		// State Change Condition
		IF (SIf.stErr.bolComError = TRUE) OR ((SIf.stErr.bolRFIDError = TRUE) AND (udiJobCount > SIf.stCfg.udiRetry)) THEN
			stStateMachine.intStateNext := cRFD_STA_Error;
		ELSIF (SIf.stErr.bolRFIDError = TRUE) THEN
			udiJobCount := udiJobCount + 1;
			stStateMachine.intStateLastCycle := 0; // Startcycle again
		ELSIF (stSubStateMachine.intState = cRFD_SUB_SubStatesEnd) THEN
			udiJobCount := 0;
			stStateMachine.intStateNext := cRFD_STA_WaitForJob;
		END_IF
		
	END_IF

//--------------------------------------------------------------------------------------
// Exit action
	IF (stStateMachine.intState<>stStateMachine.intStateNext) THEN
		SIf.intCmd := cRFD_CMD_DONE;
	END_IF
END_METHOD

METHOD PROTECTED sta_TagInitBusy : BOOL
// state implemetation
//--------------------------------------------------------------------------------------
// Entry action
	IF (stStateMachine.intState<>stStateMachine.intStateLastCycle) THEN
		stStateMachine.intStateLastCycle := stStateMachine.intState;
		
	END_IF


//--------------------------------------------------------------------------------------
// Cyclic action
	IF (stStateMachine.intState=stStateMachine.intStateLastCycle) THEN

		
		// State Change Condition
		IF (FALSE) THEN
			stStateMachine.intStateNext := cRFD_STA_Error;
		ELSIF (TRUE) THEN
			stStateMachine.intStateNext := cRFD_STA_WaitForJob;
		END_IF
		
	END_IF

//--------------------------------------------------------------------------------------
// Exit action
	IF (stStateMachine.intState<>stStateMachine.intStateNext) THEN
		IF SIf.intCmd = stStateMachine.intState THEN
			SIf.intCmd := cRFD_CMD_DONE;
		END_IF
	END_IF
END_METHOD

METHOD PROTECTED sta_WaitForJob : BOOL
// state implemetation
//--------------------------------------------------------------------------------------
// Entry action
	IF (stStateMachine.intState<>stStateMachine.intStateLastCycle) THEN
		stStateMachine.intStateLastCycle := stStateMachine.intState;
		
	END_IF


//--------------------------------------------------------------------------------------
// Cyclic action
	IF (stStateMachine.intState=stStateMachine.intStateLastCycle) THEN

		
		// State Change Condition
		IF (FALSE) THEN
			stStateMachine.intStateNext := cRFD_STA_Error;
		ELSIF (SIf.intCmd=cRFD_CMD_Read) THEN
			stStateMachine.intStateNext := cRFD_STA_ReadBusy;
		ELSIF (SIf.intCmd=cRFD_CMD_CTRL_ON) THEN
			stStateMachine.intStateNext := cRFD_STA_PowerOnBusy;
		ELSIF (SIf.intCmd=cRFD_CMD_Write) THEN
			stStateMachine.intStateNext := cRFD_STA_WriteBusy;
		ELSIF (SIf.intCmd=cRFD_CMD_MDS) THEN
			stStateMachine.intStateNext := cRFD_STA_MDSBusy;
		ELSIF (SIf.intCmd=cRFD_CMD_SLG) THEN
			stStateMachine.intStateNext := cRFD_STA_SLGBusy;
		ELSIF (SIf.intCmd=cRFD_CMD_CTRL_OFF) THEN
			stStateMachine.intStateNext := cRFD_STA_OFFBusy;
		ELSIF (SIf.intCmd=cRFD_STA_CheckBusy) THEN
			stStateMachine.intStateNext := cRFD_STA_CheckBusy;
		END_IF
		
	END_IF

//--------------------------------------------------------------------------------------
// Exit action
	IF (stStateMachine.intState<>stStateMachine.intStateNext) THEN
		;
	END_IF
END_METHOD

METHOD PROTECTED sta_WriteBusy : BOOL
// state implemetation
//--------------------------------------------------------------------------------------
// Entry action
	IF (stStateMachine.intState<>stStateMachine.intStateLastCycle) THEN
			stStateMachine.intStateLastCycle := stStateMachine.intState;
			// Byte 0 => Lenght
			aTxData[0] := 5 + SIf.stCur.usiCount;
			// Byte 1 => Command write 1=single; 11=continious
			aTxData[1] := 1;
			// Byte 2 => Spare
			aTxData[2] := 0;
			// Byte 3 => Adress MSB
			uinValue := SIf.stCur.uinAdressTag;
			uinValue := ROL(uinValue,8);
			aTxData[3] := UINT_TO_USINT(uinValue);
			// Byte 4 => Adress LSB
			aTxData[4] := UINT_TO_USINT(SIf.stCur.uinAdressTag);
			// Byte 5 =>Lenght
			aTxData[5] := SIf.stCur.usiCount;
 
			IF ((SIf.stCur.uinAdressData+SIf.stCur.usiCount <= 255) AND (SIf.stCur.usiCount+6 <= 255)) THEN
				FOR udiLoopBuffer := 0 TO (SIf.stCur.usiCount) DO
					aTxData[udiLoopBuffer+6] := SIf.stCur.pData^[SIf.stCur.uinAdressData+udiLoopBuffer];
				END_FOR	
				udiComSizeSendData := SIf.stCur.usiCount+6;
				bolComSend := TRUE;		
			ELSE
				SIf.stErr.bolComError := TRUE;
			END_IF
							
	END_IF


//--------------------------------------------------------------------------------------
// Cyclic action
	IF (stStateMachine.intState=stStateMachine.intStateLastCycle) THEN
		
		// State Change Condition
		IF (SIf.stErr.bolComError = TRUE) OR ((SIf.stErr.bolRFIDError = TRUE) AND (udiJobCount > SIf.stCfg.udiRetry)) THEN
			stStateMachine.intStateNext := cRFD_STA_Error;
		ELSIF (SIf.stErr.bolRFIDError = TRUE) THEN
			udiJobCount := udiJobCount + 1;
			stStateMachine.intStateLastCycle := 0; // Startcycle again
		ELSIF ((SIf.stErr.bolComError = 0) AND (bolWriteDone = TRUE)) THEN
			bolWriteDone := FALSE;
			udiJobCount := 0;
			stStateMachine.intStateNext := cRFD_STA_WaitForJob;
		END_IF
	
	END_IF

//--------------------------------------------------------------------------------------
// Exit action
	IF (stStateMachine.intState<>stStateMachine.intStateNext) THEN
		SIf.intCmd := cRFD_CMD_DONE;
	END_IF
END_METHOD

METHOD PROTECTED StateMachine : BOOL

// main statemachine of base controller
CASE stStateMachine.intState OF
	cRFD_STA_OffBusy: 
        THIS^.sta_OffBusy();
	cRFD_STA_Off: 
        THIS^.sta_Off();
    cRFD_STA_PowerOnBusy: 
        THIS^.sta_PowerOnBusy();
	cRFD_STA_WaitForJob: 
        THIS^.sta_WaitForJob();
	cRFD_STA_WriteBusy: 
        THIS^.sta_WriteBusy();
    cRFD_STA_ReadBusy: 
        THIS^.sta_ReadBusy();
	cRFD_STA_TagInitBusy: 
        THIS^.sta_TagInitBusy();
	cRFD_STA_CheckBusy: 
        THIS^.sta_CheckBusy();
	cRFD_STA_MDSBusy: 
        THIS^.sta_MDSBusy();
	cRFD_STA_SLGBusy: 
        THIS^.sta_SLGBusy();
    cRFD_STA_Error: 
        THIS^.sta_Error();
END_CASE;
END_METHOD

METHOD PROTECTED StateMachine_Service : BOOL


// main statemachine of base controller
CASE SIf.intServiceCmd OF
//	cRFD_CMD_MDS: 
//		THIS^.sJobWriteParameter();
//	cYAD_SCMD_READ_PARA: 
//		THIS^.sJobReadParameter();
//	cYAD_SCMD_RESET_ABSENCODER: 
//		THIS^.sJobAbsEncReset();
ELSE
	usiCaseScmd := 0;
	

	
END_CASE;
END_METHOD

END_FUNCTION_BLOCK

// POUs/Controller/Driver/RFD (RFID Driver)/FB_RFR
FUNCTION_BLOCK FB_RFR
VAR
	bolActivate: BOOL := TRUE;
	bolInitDone: BOOL;
	bolInitComDone: BOOL;
	///Communication sending is busy to the serial Card
	bolComSend: BOOL;
	/// Size of Sendingdata
	udiComSizeSendData: UDINT;
	///Communication Data Received
	bolComDataReceived: BOOL;
	/// Size of received Data from serial interface
	udiComSizeReceiveData: UDINT;
	///Sdo Setting is busy to the serial Card
	bolSdoBusy: BOOL;
	///Sdo Setting executing
	bolSdoExecute: BOOL;
	/// Job Reading is done
	bolReadDone: BOOL;
	/// Job Writing is done
	bolWriteDone: BOOL;
	/// Job Reset SLG is done
	bolResetJobDone: BOOL;
	/// Job Reset SLG has Error
	bolResetJobError: BOOL;
	/// Information to SDO Error
	udiSdoErrorNbr: UDINT;
	/// Information to Error
	udiComErrorNbr: UDINT;
	/// Count Reset cycles
	udiResetCount: UDINT;
	/// Count Job Tryals
	udiJobCount: UDINT;
	/// State information from RF ID Tag
	bytRFIDState: BYTE;
	/// BCC Calculation
	bytCheckValue: BYTE;
	/// driver specific interface
	SIf: T_RFD;
	/// get direct Buffer from Interface
	/// access over mapping!! {attribute 'TcLinkTo':='TIID^Device 1 (EtherCAT)^Box 1 (SGDV-E1 CoE Drive)^2nd Transmit PDO mapping^Status word'}
	aRxData: ARRAY[0..255] OF BYTE;
	aTxData: ARRAY[0..255] OF BYTE;
	/// Function for serial communication
	fbEcCoeSdoWrite: TC2_ETHERCAT.FB_EcCoESdoWrite;
	fbExCom: FB_ExCom;
	stStateMachine: T_RFD_StateMachine;
	stSubStateMachine: T_RFD_StateMachine;
	///case variable
	usiCase: USINT;
	///case variable for service cmd's
	usiCaseScmd: USINT;
	/// help values for parameter handling
	sinValue: SINT;
	intValue: INT;
	dinValue: DINT;
	usiValue: USINT;
	uinValue: UINT;
	udiValue: UDINT;
	uliValue: ULINT;
	pTemp: POINTER TO ARRAY[0..7] OF BYTE;
	strTemp: STRING(18);
	udiI: UDINT;
	udiLoopBuffer: UDINT;
	udiLoopData: UDINT;
	udiLoopSend: UDINT;
END_VAR

(*__________________________________________________________________________________________________
¦	
¦	Vistaprint Schweiz GmbH
¦	CH - 8401 Winterthur
¦
¦	www.vistaprint.ch - info@vistaprint.ch
¦___________________________________________________________________________________________________

Function desription:
Driver for Simatic RFID Reader RF382R 6GT2801-3AB20-0AX0 (only read function)


History:
Version		Date			Author		Comment
---------------------------------------------------------------------------------------------------
0.00.1		09.07.2013		AVME/PRE	Start history
0.00.2		18.09.2013		AVME/KVO	no initial write of parameter to RFID reader at PowerOnBusy
0.00.3		25.09.2013		AVME/KVO	always set sample error and go to error state!
___________________________________________________________________________________________________*)


IF (bolActivate) THEN // cyclic call enabled
	
	IF (bolInitDone=FALSE) THEN // first cycle -> init
		CtrlInit();
		bolInitDone := TRUE;
	ELSE
		CycleStartDuty();
		
		StateMachine_Service(); // handles asynchron service commands
		
		StateMachine();
		
		CycleEndDuty();
	END_IF
	
END_IF;

METHOD PROTECTED CtrlInit : BOOL
// one time first cyclic call
;
END_METHOD

METHOD PROTECTED CycleEndDuty : BOOL
SIf.strState := THIS^.getCmdState(intCmdState:=stStateMachine.intState,bolState:=TRUE);

IF (stStateMachine.intState<>stStateMachine.intStateNext) THEN
	stStateMachine.intState := stStateMachine.intStateNext;  // set next state for next cycle
END_IF

(***************************************************************
        Function Block Calls
***************************************************************)
END_METHOD

METHOD PROTECTED CycleStartDuty : BOOL
// ----------------------------------------------------------------------------------
// cyclic actions outside of statemachine
fbExCom(
	In_pRxData:= ADR(aRxData), 
	In_pTxData:= ADR(aTxData), 
	In_udiTxCount:= udiComSizeSendData, 
	In_bolErrorAck:= SIf.stErr.bolErrAck, 
	InOut_bolSend:= bolComSend, 
	InOut_bolRec:= bolComDataReceived, 
	Out_udiRxCount=> udiComSizeReceiveData, 
	Out_bolComError=> SIf.stErr.bolComError, 
	Out_bolProtocolErr=> SIf.stErr.bolProtcolError, 
	Out_udiErrorCode=> udiComErrorNbr);

(* program code at the beginning of each PLC cycle *)
IF bolInitComDone=TRUE THEN
	// Received Data checking and interpreting
	IF bolComDataReceived = TRUE THEN
		IF (aRxData[0] = 1) AND (udiComSizeReceiveData = 3) THEN		// Ack Reset
			IF aRxData[1] = 0 THEN
				bolResetJobDone := TRUE;
			ELSE
				 SIf.stErr.bolProtcolError := TRUE;
			END_IF
		ELSE
			// UID
			MEMCPY(destAddr:=ADR(strTemp), srcAddr:=ADR(aRxData[0]), n:=16);

			uliValue := FB_HEXSTRING_TO_ULINT(in_strSTRING:= strTemp);
			pTemp := ADR(SIf.stStatus.abyteUID[0]);
			MEMCPY(destAddr:=ADR(SIf.stStatus.abyteUID[0]), srcAddr:=ADR(uliValue), n:=8);		// COPY to ID 
			
		END_IF
		bolComDataReceived := FALSE;
	END_IF
END_IF

// always go to Error 
IF ((SIf.stErr.bolProtcolError) OR  (SIf.stErr.bolRFIDError) OR (SIf.stErr.bolSDOError)) THEN
	SIf.stErr.bolErrorActive := TRUE; // set sample Error -> got to Error state
END_IF

IF (SIf.stErr.bolErrorActive) AND (stStateMachine.intState<>cRFD_STA_Error)  THEN
	stStateMachine.intStateNext := cRFD_STA_Error;
ELSIF (stStateMachine.intState<cRFD_STA_PowerOnBusy) AND (stStateMachine.intState<>cRFD_STA_Error) THEN
	stStateMachine.intStateNext := cRFD_STA_PowerOnBusy;
END_IF

SIf.strCmd := THIS^.getCmdState(intCmdState:=SIf.intCmd,bolState:=FALSE);
END_METHOD

METHOD FB_init : BOOL
VAR_INPUT
	///if TRUE, the retain variables are initialized (warm start / cold start)
	bInitRetains: BOOL;
	///if TRUE, the instance afterwards gets moved into the copy code (online change)
	bInCopyCode: BOOL;
END_VAR
VAR
	udiTaskCnt: UDINT;
	ii: UINT;
END_VAR
SIf.intCmd := cRFD_CMD_DONE;
SIf.intServiceCmd := cRFD_CMD_DONE; // not used at the moment
stStateMachine.intStateLastCycle  := cRFD_CMD_DONE; //EntryStop of power BASE_PLC.OFF enable

// Communication Settings
SIf.stCfg.eTyp := E_Typ_RFW.RF382R;
SIf.stCfg.uinBaudrate := INT_TO_USINT(E_Typ_Baudrate.baud_38400);
SIf.stCfg.stNetId := '192.168.70.26.3.1';
SIf.stCfg.uinSlaveAddr := 1002;
END_METHOD

METHOD PROTECTED getCmdState : STRING
VAR_INPUT
	intCmdState: INT;
	bolState: BOOL;
END_VAR
// get string cmd/state string information in runtime
IF (bolState=FALSE) THEN
	// cmd's
	CASE intCmdState OF
		cRFD_CMD_DONE: 
			getCmdState := 'cRFD_CMD_DONE';
		cRFD_CMD_CTRL_ON: 
			getCmdState := 'cRFD_CMD_CTRL_ON';

	END_CASE;
ELSE

// States
	CASE intCmdState OF
		cRFD_STA_Error: 
			getCmdState := 'cRFD_STA_Error';
		cRFD_STA_WaitForJob: 
			getCmdState := 'cRFD_STA_WaitForJob';
		cRFD_STA_PowerOnBusy: 
			getCmdState := 'cRFD_STA_PowerOnBusy';

	END_CASE;
END_IF
END_METHOD

METHOD getSIf : POINTER TO T_RFD
getSIf := ADR(SIf);
END_METHOD

METHOD PROTECTED sta_Error : BOOL
// state implemetation
//--------------------------------------------------------------------------------------
// Entry action
	IF (stStateMachine.intState<>stStateMachine.intStateLastCycle) THEN
		stStateMachine.intStateHistory := stStateMachine.intStateLastCycle;
		stStateMachine.intStateLastCycle := stStateMachine.intState;
		
	END_IF


//--------------------------------------------------------------------------------------
// Cyclic action
	IF (stStateMachine.intState=stStateMachine.intStateLastCycle) THEN
		SIf.stErr.bolErrorActive := TRUE;
		IF (SIf.stErr.bolComError = TRUE) OR (SIf.stErr.bolProtcolError = TRUE) THEN
			SIf.stErr.udiErrorID := udiComErrorNbr;
		ELSIF SIf.stErr.bolSDOError = TRUE THEN
			SIf.stErr.udiErrorID := udiSdoErrorNbr;
		ELSIF (udiResetCount >=SIf.stCfg.udiRetry) OR (udiJobCount >= SIf.stCfg.udiRetry) THEN
			SIf.stErr.udiErrorID := SIf.stCfg.udiRetry;
		ELSE
			SIf.stErr.udiErrorID := 0;
		END_IF

		
		// State Change Condition
		IF (SIf.stErr.bolErrAck = TRUE) THEN
			// Reset all active errors
			SIf.stErr.bolErrorActive := FALSE;
			SIf.stErr.bolComError := FALSE;
			SIf.stErr.bolProtcolError := FALSE;
			SIf.stErr.bolSDOError := FALSE;
			SIf.stErr.udiErrorID := 0;
			stStateMachine.intStateNext := cRFD_STA_PowerOnBusy;		
		END_IF
	END_IF




//--------------------------------------------------------------------------------------
// Exit action
	IF (stStateMachine.intState<>stStateMachine.intStateNext) THEN
		;
	END_IF
END_METHOD

METHOD PROTECTED sta_PowerOnBusy : BOOL
// state implemetation
//--------------------------------------------------------------------------------------
// Entry action
	IF (stStateMachine.intState<>stStateMachine.intStateLastCycle) THEN
		stStateMachine.intStateLastCycle := stStateMachine.intState;
			//IF bolInitComDone=FALSE THEN
				// direct write parameter doesn't work!! KVO 17.09.2013 with new Kannegiesser RFID
				// Feedback rx[0..2] 255 4 251 -> Baudrate/task time not 2ms
				// no Feedback -> parameter set? estimated  rx[0..2] 1 0 1
				// decision with Rolf Engelputzeder 18.09.2013 
				// don't use write parameter at the moment:
				stSubStateMachine.intState := cRFD_SUB_SubStatesEnd;// cRFD_SUB_ClearBuffer;		// First Time set Baudrate and communication Settings
				stSubStateMachine.intStateNext := cRFD_SUB_SubStatesEnd;// cRFD_SUB_ClearBuffer;		// First Time set Baudrate and communication Settings
				bolInitComDone := TRUE; // old without this condition
				
				(*
				// original set parameter to RFID
				stSubStateMachine.intState := cRFD_SUB_ClearBuffer;		// First Time set Baudrate and communication Settings
				stSubStateMachine.intStateNext := cRFD_SUB_ClearBuffer;
				*)
			//END_IF
			bolSdoExecute := FALSE;
			bolResetJobDone := FALSE;
	END_IF


//--------------------------------------------------------------------------------------
// Cyclic action
	IF (stStateMachine.intState=stStateMachine.intStateLastCycle) THEN
		
		// main statemachine of base controller
		CASE stSubStateMachine.intState OF
			cRFD_SUB_SetBaudrate:
				IF stSubStateMachine.intStateLastCycle <> stSubStateMachine.intState THEN
					stSubStateMachine.intStateLastCycle := stSubStateMachine.intState;
				END_IF
				fbEcCoeSdoWrite(
					sNetId:= SIf.stCfg.stNetId, 
					nSlaveAddr:= SIf.stCfg.uinSlaveAddr, 
					nIndex:= SIf.stCfg.uinCoeIndexComSettings, 
					nSubIndex:= SIf.stCfg.usiCoeSubindexComBaudrate, 
					pSrcBuf:= ADR(SIf.stCfg.uinBaudrate), 
					cbBufLen:= SIZEOF(SIf.stCfg.uinBaudrate), 
					bExecute:= bolSdoExecute, 
					tTimeout:= DEFAULT_ADS_TIMEOUT, 
					bBusy=> bolSdoBusy, 
					bError=> SIf.stErr.bolSDOError, 
					nErrId=> udiSdoErrorNbr);
					
					
				IF 	(bolSdoExecute = TRUE) THEN
					IF ((SIf.stErr.bolSDOError = FALSE) AND (bolSdoBusy = FALSE)) THEN
						bolSdoExecute := FALSE;
						stSubStateMachine.intStateNext := cRFD_SUB_ClearBuffer;
					END_IF
				ELSE
					bolSdoExecute := TRUE;
				END_IF
				
			
			cRFD_SUB_SetComSettings:
				IF stSubStateMachine.intStateLastCycle <> stSubStateMachine.intState THEN
					stSubStateMachine.intStateLastCycle := stSubStateMachine.intState;
				END_IF
				fbEcCoeSdoWrite(
					sNetId:= SIf.stCfg.stNetId, 
					nSlaveAddr:= SIf.stCfg.uinSlaveAddr, 
					nSubIndex:= SIf.stCfg.usiCoeSubindexComDataframe, 
					nIndex:= SIf.stCfg.uinCoeIndexComSettings, 
					pSrcBuf:= ADR(SIf.stCfg.uinComSettings), 
					cbBufLen:= SIZEOF(SIf.stCfg.uinComSettings), 
					bExecute:= bolSdoExecute, 
					tTimeout:= T#2S, 
					bBusy=> bolSdoBusy, 
					bError=> SIf.stErr.bolSDOError, 
					nErrId=> udiSdoErrorNbr);
					
				IF 	(bolSdoExecute = TRUE) THEN
					IF ((SIf.stErr.bolSDOError = FALSE) AND (bolSdoBusy = FALSE)) THEN
						bolSdoExecute := FALSE;
						stSubStateMachine.intStateNext := cRFD_SUB_ClearBuffer;
					END_IF
				ELSE
					bolSdoExecute := TRUE;
				END_IF

	
			cRFD_SUB_ClearBuffer: 	 
				IF stSubStateMachine.intStateLastCycle <> stSubStateMachine.intState THEN
					stSubStateMachine.intStateLastCycle := stSubStateMachine.intState;
				END_IF
				bolInitComDone := TRUE;
				IF (SIf.stErr.bolComError = FALSE) THEN
					stSubStateMachine.intStateNext := cRFD_SUB_InitString;
				END_IF

				
			cRFD_SUB_InitString: 
				IF stSubStateMachine.intStateLastCycle <> stSubStateMachine.intState THEN
					stSubStateMachine.intStateLastCycle := stSubStateMachine.intState;
					// Byte 0 => Para = 16#01
					aTxData[0] := 1;
					// Byte 1 => Memory
					aTxData[1] := SIf.stCfg.usiMemory;
					// Byte 2 => Spare
					aTxData[2] := 0;
					// Byte 3 => Spare
					aTxData[3] := 0;
					// Byte 4 => Spare
					aTxData[4] := 0;
					// Byte 5 => Spare
					aTxData[5] := 0;
					// Byte 6 => Spare
					aTxData[6] := 0;
					// Byte 7 => Scan Mode
					aTxData[7] := SIf.stCfg.usiScanMode;
					// Byte 8 => Lock Time High Byte
					aTxData[8] := UINT_TO_BYTE(SIf.stCfg.uinLockTime_ms/100);
					// Byte 9 => Lock Time Low Byte
					aTxData[9] := UINT_TO_BYTE(SHR((SIf.stCfg.uinLockTime_ms/100),8));
					// Byte 10 => Spare
					aTxData[10] := 0;
					// Byte 11 => Spare
					aTxData[11] := 0;
					// Byte 12 => Spare
					aTxData[12] := 0;
					// Byte 13 => Spare
					aTxData[13] := 0;
					// Byte 14 => Spare
					aTxData[14] := 0;
					// Byte 15 => Spare
					aTxData[15] := 0;
					// Byte 16 => Spare
					aTxData[16] := 0;
					// Byte 17 => Spare
					aTxData[17] := 0;
					// Byte 18 => Spare
					aTxData[18] := 0;
					// Byte 19 => Spare
					aTxData[19] := 0;
					// Byte 20 => Spare
					aTxData[20] := 0;
					// Byte 21 => Spare
					aTxData[21] := 0;
					// Byte 22 => Spare
					aTxData[22] := 0;

					bytCheckValue := aTxData[0] XOR aTxData[1];
					FOR udiI := 2 TO  22 DO
						bytCheckValue := bytCheckValue XOR aTxData[udiI];
					END_FOR
					
					// Byte 23 => BCC
					aTxData[23] := bytCheckValue;
					
					udiComSizeSendData := 24;
					bolComSend := TRUE;
				END_IF
			
				IF ((SIf.stErr.bolComError = 0) AND (bolComSend = FALSE)) THEN	
					stSubStateMachine.intStateNext := cRFD_SUB_CheckPon;
				END_IF

			cRFD_SUB_CheckPon:
				IF (bolResetJobDone = TRUE) THEN
					stSubStateMachine.intStateNext := cRFD_SUB_SubStatesEnd;
				ELSIF (bolResetJobError =TRUE) AND (udiResetCount < SIf.stCfg.udiRetry) THEN
					bolResetJobError := FALSE;
					udiResetCount := udiResetCount + 1;
					stSubStateMachine.intStateNext := cRFD_SUB_InitString;
				END_IF
				
			cRFD_SUB_SubStatesEnd:
				;
		END_CASE
		
		stSubStateMachine.intStateLastCycle := stSubStateMachine.intState;
		IF (stSubStateMachine.intState<>stSubStateMachine.intStateNext) THEN
			stSubStateMachine.intState := stSubStateMachine.intStateNext;  // set next state for next cycle
		END_IF
		

		// State Change Condition
		IF (SIf.stErr.bolComError = TRUE) OR (SIf.stErr.bolSDOError = TRUE) OR (udiResetCount >= SIf.stCfg.udiRetry) THEN
			stStateMachine.intStateNext := cRFD_STA_Error;
		ELSIF (stSubStateMachine.intStateNext = cRFD_SUB_SubStatesEnd) THEN
			stStateMachine.intStateNext := cRFD_STA_WaitForJob;
		END_IF
		
	END_IF


//--------------------------------------------------------------------------------------
// Exit action
	IF (stStateMachine.intState<>stStateMachine.intStateNext) THEN
		SIf.intCmd := cRFD_CMD_DONE;
		SIf.stStatus.bolStartupOk := TRUE;
	END_IF
END_METHOD

METHOD PROTECTED sta_WaitForJob : BOOL
// state implemetation
//--------------------------------------------------------------------------------------
// Entry action
	IF (stStateMachine.intState<>stStateMachine.intStateLastCycle) THEN
		stStateMachine.intStateLastCycle := stStateMachine.intState;
		
	END_IF


//--------------------------------------------------------------------------------------
// Cyclic action
	IF (stStateMachine.intState=stStateMachine.intStateLastCycle) THEN

		
		// State Change Condition
		IF (SIf.intCmd=cRFD_CMD_CTRL_ON) THEN
			stStateMachine.intStateNext := cRFD_STA_PowerOnBusy;
		END_IF
		
	END_IF

//--------------------------------------------------------------------------------------
// Exit action
	IF (stStateMachine.intState<>stStateMachine.intStateNext) THEN
		;
	END_IF
END_METHOD

METHOD PROTECTED StateMachine : BOOL

// main statemachine of base controller
CASE stStateMachine.intState OF
    cRFD_STA_PowerOnBusy: 
        THIS^.sta_PowerOnBusy();
	cRFD_STA_WaitForJob: 
        THIS^.sta_WaitForJob();
   cRFD_STA_Error: 
        THIS^.sta_Error();
END_CASE;
END_METHOD

METHOD PROTECTED StateMachine_Service : BOOL


// main statemachine of base controller
CASE SIf.intServiceCmd OF

ELSE
	usiCaseScmd := 0;
	

	
END_CASE;
END_METHOD

END_FUNCTION_BLOCK

// POUs/Controller/Lvl0/BCC (Barcode controller)/FB_BCC
FUNCTION_BLOCK FB_BCC EXTENDS FB_CtrlBase
VAR_INPUT
	In_bolSensorTrigScan: BOOL;
	pBCD_SIf_In: POINTER TO T_BCD;
END_VAR
VAR
	/// Specific interface struct for public access
	SIf: T_Ctrl_SIf_BCC;
	/// old barcode to know that a new barcode is present from sensor
	uliBarCodeOld: ULINT;
	/// simulated barcode
	uliSimBarCode: ULINT;
	/// Variables for driver simulation
	pBCD_SIf: POINTER TO T_BCD;
	stBCD_Sim: T_BCD;
	/// Edge detection of trigger sensor 
	bolSensorTrigScanOld: BOOL;
	/// Exceute scan flag
	bolExecuteScan: BOOL;
	udiScanDelayTimer_ms: UDINT;
END_VAR

(*__________________________________________________________________________________________________
¦	
¦	Vistaprint Schweiz GmbH
¦	CH - 8401 Winterthur
¦
¦	www.vistaprint.ch - info@vistaprint.ch
¦___________________________________________________________________________________________________

Function desription:
Barcode reader controller.
Controls the communication to the barcode reader.

History:
Version		Date			Author		Comment
---------------------------------------------------------------------------------------------------
0.00.1		06.01.2014		AVME/DSC	Start history
0.00.2		07.01.2014		AVME/DSC	Basic functionalities implemented and tested. 	
0.00.3		27.01.2014		AVME/DSC	- Added info "bolNoRead" in cur interface
					 					- Revision in error recovery
0.00.4		15.07.2014		AVME/DSC   RP-208 - Implement sensor signal input for triggering a barcode scan
									   The controller is already implemented with a common interface waiting for command READ to execute a new barcode scan.
									   Controller is now equipped with a further option to execute a scan by checking a sensor signal input.
0.00.5		24.10.2014		HLV/MAH		driver can be used for Sick or Keyence scanner configured by SIf.Cfg.iSensorType := E_BCD_Type.xxxx
										the port of Keyence scanner must be always 9004
										if Keyence scanner is used, FB_SocketCloseAll must be called in main PRG (see MiddlePRG in BaseElementsSample)

___________________________________________________________________________________________________*)

SUPER^();

(*
IF (me.bolActivate) AND (pBCD_SIf_In<>0) THEN // cyclic call enabled
	IF (CIf.Info.bolInitDone=FALSE) THEN // first cycle -> init
		CtrlInit();
		CIf.Info.bolInitDone := TRUE;
	ELSE
		CycleStartDuty();
	
		Always();
		
		StateMachine();
		
		CycleEndDuty();
	
	END_IF
END_IF;
*)

{attribute 'object_name' := 'Always'}
METHOD PROTECTED Always : BOOL
SUPER^.Always();

// Simulation
IF (CIf.SwCfg.bolSimulation) THEN
	// Access to driver empty structure
	pBCD_SIf := ADR(stBCD_Sim);
ELSE
	// Access to real driver interface
	pBCD_SIf := pBCD_SIf_In;
END_IF

// ----------------------------------------------------------------------------------
// cyclic actions outside of statemachine
IF (me.StateMachine.intState<>cSTA_SINGLE_ANSWER) THEN
	
	// Handle sensor trigger input
	// --------------------------------------------
	// Check pos. edge of the sensor 
	IF (SIf.In.bolSensorTrigScan.intern) AND NOT (bolSensorTrigScanOld) THEN	
		// Kick-off a new scan
		bolExecuteScan:= TRUE;
	END_IF

	// Execute scan?
	IF (bolExecuteScan) AND (me.StateMachine.intState<>BCC_CmdState.cBCC_STA_READBusy) THEN
		// Wait X-time (time delay) before executing a barcode scan 
		IF (udiScanDelayTimer_ms >= SIf.Par.udiExecuteScanDelayTime_ms) THEN
			bolExecuteScan:= FALSE;
			me.StateMachine.intStateNext := BCC_CmdState.cBCC_STA_READBusy;
		END_IF
		// Timer handling
		udiScanDelayTimer_ms:= udiScanDelayTimer_ms + me.FUBInfo.udiSample_ms;
	ELSE
		// Reset timer
		udiScanDelayTimer_ms:= 0;
	END_IF
	
	// Check trigger error conditions
	// --------------------------------------------
	// In case if a new scan will be triggered by the sensor trigger input but a scan is already in progress -> set warning!
	// Check if Scan in progress
	IF (me.StateMachine.intState=BCC_CmdState.cBCC_STA_READBusy) THEN
		// New pos. trigger signal detected during scan
		IF (SIf.In.bolSensorTrigScan.intern) AND (bolSensorTrigScanOld <> SIf.In.bolSensorTrigScan.intern) THEN
			// SIf.Alm[6].strText := 'New scan was triggered during a scan was already in progress. Check line speed and barcode reader settings!';
			pfbAlarmCtrl^.setAlarm(CIf.Info.intCtrlId,6,0,ADR(SIf.Alm),E_AlmState.RST,CIf.Job.eMe_ActivAlmClass);	
		END_IF
	END_IF
	
	// Save sensor signal. Used for edge detection
	bolSensorTrigScanOld:= SIf.In.bolSensorTrigScan.intern;
		
	// Status info from driver
	// --------------------------------------------
	SIf.Cur.bolComChecked:= pBCD_SIf^.stStatus.bolComChecked;
	SIf.Cur.bolConnected:= pBCD_SIf^.stStatus.bolSocketConnected;
	
END_IF

// config driver
pBCD_SIf^.stCfg.bolSimulation := CIf.SwCfg.bolSimulation;
pBCD_SIf^.stCfg.strSensorIPAdr := SIf.Cfg.strSensorIPAdr;
pBCD_SIf^.stCfg.udiSensorPort := SIf.Cfg.udiSensorPort;
pBCD_SIf^.stCfg.iSensorType := SIf.Cfg.iSensorType;

// ----------------------------------------------------------------------------------
// Always change actions in Base Library
// ----------------------------------------------------------------------------------
// overrule error always from base -> no EOFF State!! in EOFF go to OFF
IF (me.StateMachine.intStateNext = cSTA_EOFFBusy) THEN
	IF (me.StateMachine.intState=cSTA_OFF) THEN
		me.StateMachine.intStateNext := cSTA_OFF;
	ELSE // stay in OFF
		me.StateMachine.intStateNext := cSTA_OFFBusy;
	END_IF
END_IF

// Conditions Always
IF (((me.Alarm.eActivAlmClass=E_AlmClass.EOFF) OR (me.Alarm.eActivAlmClass=E_AlmClass.OFF) OR (me.intCmd=cCMD_OFF))
		 AND (me.StateMachine.intState<>cSTA_ERROR) AND (me.StateMachine.intState<>cSTA_ERRORQuit) AND
		(me.StateMachine.intState<>cSTA_OFF) AND (me.StateMachine.intState<>cSTA_OFFBusy)) THEN
	// alarm evt EOFF, OFF or cmd off
	me.StateMachine.intStateNext := cSTA_OFFBusy;
END_IF
END_METHOD

{attribute 'object_name' := 'FB_init'}
METHOD FB_init : BOOL
VAR_INPUT
	///if TRUE, the retain variables are initialized (warm start / cold start)
	bInitRetains: BOOL;
	///if TRUE, the instance afterwards gets moved into the copy code (online change)
	bInCopyCode: BOOL;
END_VAR
VAR
	udiTaskCnt: UDINT;
	ii: UINT;
END_VAR
//------------------------------------------------------------------------------------------------------------------------
// to manually change in new FUB implementation!!!
// define valid commands for this controller
FOR ii:= 0 TO (SIZEOF(CIf.Job.aCmdList)/SIZEOF(CIf.Job.aCmdList[0])-1) BY 1 DO
	IF (CIf.Job.aCmdList[ii].intCmd=cCMD_INITIALIZED) THEN
		// found first empty array element
		EXIT;
	END_IF
END_FOR
CIf.Job.aCmdList[ii].intCmd := cBCC_CMD_READ;
CIf.Job.aCmdList[ii].strName := 'Read'; 
CIf.Job.aCmdList[ii].bolAvailable := TRUE;

// set name of class/typ
CIf.Info.strType := 'FB_BCC';
CIf.Info.strFullName := 'Barcode Controller';

// set alarm class
SIf.Alm[1].eAlmClass := E_AlmClass.INFO;
SIf.Alm[1].strText := 'Barcode reader driver error'; 
SIf.Alm[2].eAlmClass := E_AlmClass.OFF;
SIf.Alm[2].strText := 'Initialisation error from barcode reader. No answer from device.';
SIf.Alm[3].eAlmClass := E_AlmClass.INFO;
SIf.Alm[3].strText := 'Barcode could not be read. Answer *NoRead* from device';
SIf.Alm[4].eAlmClass := E_AlmClass.INFO;
SIf.Alm[4].strText := 'Timeout wait on data';
SIf.Alm[5].eAlmClass := E_AlmClass.INFO;
SIf.Alm[5].strText := 'Error response from sensor';
SIf.Alm[6].eAlmClass := E_AlmClass.WARNING;
SIf.Alm[6].strText := 'New scan was triggered during a scan was already in progress!';

//*******************************************************************************
// initial values
//*******************************************************************************

// software configuration
CIf.SwCfg.bolExist := TRUE;
CIf.SwCfg.bolSimulation := FALSE;

// parameter
SIf.Par.udiTORead_ms := 4000;  		// Has to be correspond with the "duration" setting of sensor object trigger
SIf.Par.udiTOPowerOn_ms := 3000;
SIf.Par.udiExecuteScanDelayTime_ms:= 500;

// configuration
SIf.Cfg.strSensorIPAdr := '192.168.1.103';
SIf.Cfg.udiSensorPort := 9004;
SIf.Cfg.iSensorType := E_BCD_Type.KEYENCE;

// simulation
uliSimBarCode:= 1250000000000;
END_METHOD

{attribute 'object_name' := 'getCmdState'}
METHOD PROTECTED getCmdState : STRING
VAR_INPUT
	intCmdState: INT;
	bolState: BOOL;
END_VAR
getCmdState := SUPER^.getCmdState(intCmdState:=intCmdState,bolState:=bolState); // get global/base defined cmds/states
IF (getCmdState='') THEN // global not defined get local
	// get string cmd/state string information in runtime
	IF (bolState=FALSE) THEN
		// cmd's
		CASE intCmdState OF
			cBCC_CMD_READ: 
				getCmdState := 'READ';
		END_CASE;
	ELSE
	
	// cmd's
		CASE intCmdState OF
			cBCC_STA_READBusy: 
				getCmdState := 'READBusy';
			cBCC_STA_READ: 
				getCmdState := 'READ';
		END_CASE;
	END_IF
END_IF
END_METHOD

{attribute 'object_name' := 'getCtrlSIf'}
METHOD getCtrlSIf : POINTER TO T_Ctrl_SIf_BCC
getCtrlSIf := ADR(SIf);
END_METHOD

{attribute 'object_name' := 'IoInBridge'}
METHOD PROTECTED IoInBridge : BOOL
// digitale and analoge inputs read from hardware or forcing
SIf.In.bolSensorTrigScan.map := THIS^.In_bolSensorTrigScan;

IF (CIf.SwCfg.bolSimulation = FALSE) THEN
	getInBol(CIf.Job.bolIoForce,ADR(SIf.In.bolSensorTrigScan));
ELSE
	//simulation of global IO
END_IF
END_METHOD

{attribute 'object_name' := 'IoOutBridge'}
METHOD PROTECTED IoOutBridge : BOOL
// digitale and analoge inputs read from hardware or forcing
IF (CIf.SwCfg.bolSimulation = FALSE) THEN
	// check interlocks to prevent damages
	IF (CIf.Job.bolIlkOverwrite=FALSE) THEN
		;
		// no physical outputs
	END_IF
END_IF
END_METHOD

{attribute 'object_name' := 'sta_ERROR'}
METHOD PROTECTED sta_ERROR : BOOL
// state implemetation
//--------------------------------------------------------------------------------------
// Entry action
	IF (me.StateMachine.intState<>me.StateMachine.intStateLastCycle) THEN
		me.StateMachine.intStateHistory := me.StateMachine.intStateLastCycle; // -> possibillity to go back to state before error
		me.StateMachine.intStateLastCycle := me.StateMachine.intState;
		
		// Driver error activ
		IF (pBCD_SIf^.stErr.bolErrorActive = TRUE) THEN
			// SIf.Alm[1].strText := 'Barcode reader driver error'; 
			pfbAlarmCtrl^.setAlarm(CIf.Info.intCtrlId,1,UDINT_TO_DINT(pBCD_SIf^.stErr.udiErrorID),ADR(SIf.Alm),E_AlmState.RST,CIf.Job.eMe_ActivAlmClass);
			// Error response from sensor
			IF (pBCD_SIf^.stErr.bolSensorError = TRUE) THEN
				// SIf.Alm[5].strText := 'Error response from sensor with sopas error number';
				pfbAlarmCtrl^.setAlarm(CIf.Info.intCtrlId,5,UDINT_TO_DINT(pBCD_SIf^.stErr.udiErrorID),ADR(SIf.Alm),E_AlmState.RST,CIf.Job.eMe_ActivAlmClass);		
			END_IF
		ELSE
			// Close TCP socket		
			pBCD_SIf^.intCmd := cBCD_CMD_CLOSE_SOCKET;  	
		END_IF
		
	END_IF

//--------------------------------------------------------------------------------------
// Cyclic action
	IF (me.StateMachine.intState=me.StateMachine.intStateLastCycle) THEN
	
		// State Change Condition
		IF (CIf.Job.bolAlmReset = TRUE) THEN
			// Error ack driver 
			pBCD_SIf^.stErr.bolErrAck:= TRUE;
			me.StateMachine.intStateNext := cSTA_ERRORQuit;
		END_IF
	END_IF

//--------------------------------------------------------------------------------------
// Exit action
	IF (me.StateMachine.intState<>me.StateMachine.intStateNext) THEN
		;
	END_IF
END_METHOD

{attribute 'object_name' := 'sta_OFF'}
METHOD PROTECTED sta_OFF : BOOL
// state implemetation
//--------------------------------------------------------------------------------------
// Entry action
	IF (me.StateMachine.intState<>me.StateMachine.intStateLastCycle) THEN
		me.StateMachine.intStateLastCycle := me.StateMachine.intState;
		
	END_IF


//--------------------------------------------------------------------------------------
// Cyclic action
	IF (me.StateMachine.intState=me.StateMachine.intStateLastCycle) THEN
		
		;		
		// State Change Condition
		IF (me.Alarm.eActivAlmClass<>E_AlmClass.EOFF) AND (me.Alarm.eActivAlmClass<>E_AlmClass.OFF) THEN	
			IF(me.intCmd=cBCC_CMD_READ) THEN
				me.StateMachine.intStateNext := cBCC_STA_READBusy;
			END_IF
		END_IF
	END_IF

//--------------------------------------------------------------------------------------
// Exit action
	IF (me.StateMachine.intState<>me.StateMachine.intStateNext) THEN
		;
	END_IF
END_METHOD

{attribute 'object_name' := 'sta_OFFBusy'}
METHOD PROTECTED sta_OFFBusy : BOOL
// state implemetation
//--------------------------------------------------------------------------------------
// Entry action
	IF (me.StateMachine.intState<>me.StateMachine.intStateLastCycle) THEN
		me.StateMachine.intStateLastCycle := me.StateMachine.intState;
		
		// Simulation timer	
		fbSimulationTimer.IN := FALSE;
		fbSimulationTimer.PT := UDINT_TO_TIME(SIf.Par.udiTORead_ms / 2);
		fbSimulationTimer(); // set time/reset timer
		fbSimulationTimer.IN := TRUE; // start timer
		
	END_IF

//--------------------------------------------------------------------------------------
// Cyclic action
	IF (me.StateMachine.intState=me.StateMachine.intStateLastCycle) THEN
		
		// Simulation
		IF (CIf.SwCfg.bolSimulation) THEN
			fbSimulationTimer(); // simulation time
			IF (fbSimulationTimer.Q) THEN
				pBCD_SIf^.intCmd := cBCD_CMD_DONE;
			END_IF
		END_IF
			
		// State Change Condition
		IF (pBCD_SIf^.stErr.bolErrorActive = TRUE) THEN
			me.StateMachine.intStateNext :=  cSTA_ERROR;
		ELSIF(pBCD_SIf^.intCmd = cBCD_CMD_DONE) THEN
			me.StateMachine.intStateNext := cSTA_OFF;
		END_IF
	END_IF

//--------------------------------------------------------------------------------------
// Exit action
	IF (me.StateMachine.intState<>me.StateMachine.intStateNext) THEN
		;
	END_IF
END_METHOD

{attribute 'object_name' := 'sta_PON'}
METHOD PROTECTED sta_PON : BOOL
// state implemetation
//--------------------------------------------------------------------------------------
// Entry action
	IF (me.StateMachine.intState<>me.StateMachine.intStateLastCycle) THEN
		me.StateMachine.intStateLastCycle := me.StateMachine.intState;
		
	END_IF


//--------------------------------------------------------------------------------------
// Cyclic action
	IF (me.StateMachine.intState=me.StateMachine.intStateLastCycle) THEN
		
		;	
		// State Change Condition
		me.StateMachine.intStateNext := cSTA_OFFBusy;
	END_IF


//--------------------------------------------------------------------------------------
// Exit action
	IF (me.StateMachine.intState<>me.StateMachine.intStateNext) THEN
		;
	END_IF
END_METHOD

{attribute 'object_name' := 'sta_PONBusy'}
METHOD PROTECTED sta_PONBusy : BOOL
// state implemetation
//--------------------------------------------------------------------------------------
// Entry action
	IF (me.StateMachine.intState<>me.StateMachine.intStateLastCycle) THEN
		me.StateMachine.intStateLastCycle := me.StateMachine.intState;
		
		// Simulation timer	
		fbSimulationTimer.IN := FALSE;
		fbSimulationTimer.PT := UDINT_TO_TIME(SIf.Par.udiTORead_ms / 2);
		fbSimulationTimer(); // set time/reset timer
		fbSimulationTimer.IN := TRUE; // start timer
		
		// Reset driver status
		pBCD_SIf^.stStatus.bolSocketConnected := FALSE;
		pBCD_SIf^.stStatus.bolComChecked := FALSE;
	END_IF

//--------------------------------------------------------------------------------------
// Cyclic action
	IF (me.StateMachine.intState=me.StateMachine.intStateLastCycle) THEN
			
		// Simulation
		IF (CIf.SwCfg.bolSimulation) THEN
			fbSimulationTimer(); // simulation time
			IF (fbSimulationTimer.Q) THEN
				// Set driver status
				pBCD_SIf^.stStatus.bolSocketConnected := TRUE;
				pBCD_SIf^.stStatus.bolComChecked := TRUE;		
			END_IF
		END_IF
			
		// Try to open the TCP socket
		IF (pBCD_SIf^.stStatus.bolSocketConnected = FALSE) THEN		
			pBCD_SIf^.intCmd := cBCD_CMD_CONNECT_SOCKET; 
		END_IF 
					
		// Check if socket connected
		IF (pBCD_SIf^.stStatus.bolSocketConnected = TRUE) AND (pBCD_SIf^.stStatus.bolComChecked = FALSE) THEN
			pBCD_SIf^.intCmd :=	cBCD_CMD_COM_TEST; // Execute a communication test to see if the device answer		
		END_IF
		
		// State Change Condition
		IF ((pBCD_SIf^.stErr.bolErrorActive = TRUE) OR (me.StateMachine.udiTimeInState_ms >= SIf.Par.udiTOPowerOn_ms)) THEN
			// SIf.Alm[2].strText := 'Initialisation error from barcode reader. No answer from device.';
			pfbAlarmCtrl^.setAlarm(CIf.Info.intCtrlId,2,0,ADR(SIf.Alm),E_AlmState.RST,CIf.Job.eMe_ActivAlmClass);
			me.StateMachine.intStateNext := cSTA_ERROR;				
		ELSIF (pBCD_SIf^.stStatus.bolComChecked = TRUE) THEN
			me.StateMachine.intStateNext := cSTA_PON;
		END_IF
	END_IF

//--------------------------------------------------------------------------------------
// Exit action
	IF (me.StateMachine.intState<>me.StateMachine.intStateNext) THEN
		;
	END_IF
END_METHOD

{attribute 'object_name' := 'sta_READ'}
METHOD PROTECTED sta_READ : BOOL
// state implemetation
//--------------------------------------------------------------------------------------
// Entry action
	IF (me.StateMachine.intState<>me.StateMachine.intStateLastCycle) THEN
		me.StateMachine.intStateLastCycle := me.StateMachine.intState;

	END_IF

//--------------------------------------------------------------------------------------
// Cyclic action
	IF (me.StateMachine.intState=me.StateMachine.intStateLastCycle) THEN

		// Simulation
		IF (CIf.SwCfg.bolSimulation) THEN
			;
		END_IF
		
		// State Change Condition
		IF(me.intCmd=cBCC_CMD_READ) THEN
			me.StateMachine.intStateNext := cBCC_STA_READBusy;
		END_IF
	END_IF

//--------------------------------------------------------------------------------------
// Exit action
	IF (me.StateMachine.intState<>me.StateMachine.intStateNext) THEN
		;
	END_IF
END_METHOD

{attribute 'object_name' := 'sta_READBusy'}
METHOD PROTECTED sta_READBusy : BOOL
// state implemetation
//--------------------------------------------------------------------------------------
// Entry action
	IF (me.StateMachine.intState<>me.StateMachine.intStateLastCycle) THEN
		me.StateMachine.intStateLastCycle := me.StateMachine.intState;
		
		// Simulation timer	
		fbSimulationTimer.IN := FALSE;
		fbSimulationTimer.PT := UDINT_TO_TIME(SIf.Par.udiTORead_ms / 2);
		fbSimulationTimer(); // set time/reset timer
		fbSimulationTimer.IN := TRUE; // start timer
		
		// Init
		SIf.Cur.bolNewCodeReaded:= FALSE;
		SIf.Cur.bolNoRead:= FALSE;
		SIf.Cur.stData.uliBarCode:= 0;
		SIf.Cur.stData.strBarCode:= '';
		
		// Read barcode
		pBCD_SIf^.intCmd := cBCD_CMD_READ_BARCODE;
	END_IF


//--------------------------------------------------------------------------------------
// Cyclic action
	IF (me.StateMachine.intState=me.StateMachine.intStateLastCycle) THEN

		// Simulation
		IF (CIf.SwCfg.bolSimulation) THEN
			fbSimulationTimer(); // simulation time
			IF (fbSimulationTimer.Q) THEN
				SIf.Cur.bolNewCodeReaded:= TRUE;
				uliSimBarCode:= uliSimBarCode + 1;
				pBCD_SIf^.stData.uliBarCode:= uliSimBarCode;
				pBCD_SIf^.stData.strBarCode:= ULINT_TO_STRING(pBCD_SIf^.stData.uliBarCode);
				pBCD_SIf^.intCmd := cBCD_CMD_DONE;		
			END_IF
		END_IF	

		// Check for new barcode
		IF (pBCD_SIf^.stData.uliBarCode <> uliBarCodeOld) AND (pBCD_SIf^.stData.uliBarCode<>0) THEN
			uliBarCodeOld:= pBCD_SIf^.stData.uliBarCode;
			SIf.Cur.bolNewCodeReaded:= TRUE;
		END_IF
		
		// Get data from driver
		SIf.Cur.stData.uliBarCode:= pBCD_SIf^.stData.uliBarCode;
		SIf.Cur.stData.strBarCode:= pBCD_SIf^.stData.strBarCode;			
		
		// State Change Condition
		IF (pBCD_SIf^.stErr.bolErrorActive = TRUE) THEN  
			me.StateMachine.intStateNext :=  cSTA_ERROR;
		ELSIF (me.StateMachine.udiTimeInState_ms > SIf.Par.udiTORead_ms) THEN
			// SIf.Alm[4].strText := 'Timeout wait on data';
			pfbAlarmCtrl^.setAlarm(CIf.Info.intCtrlId,4,0,ADR(SIf.Alm),E_AlmState.RST,CIf.Job.eMe_ActivAlmClass);
			me.StateMachine.intStateNext :=  cSTA_ERROR;
		ELSIF (pBCD_SIf^.intCmd = cBCD_CMD_DONE) THEN
			IF (SIf.Cur.stData.uliBarCode=0) THEN
				SIf.Cur.bolNoRead:= TRUE;
				uliBarCodeOld:= 0;
				// SIf.Alm[3].strText := 'Barcode could not be read. Answer *NoRead* from device';
				pfbAlarmCtrl^.setAlarm(CIf.Info.intCtrlId,3,0,ADR(SIf.Alm),E_AlmState.RST,CIf.Job.eMe_ActivAlmClass);	
			END_IF		
			me.StateMachine.intStateNext := cBCC_STA_READ;
		END_IF
	END_IF

//--------------------------------------------------------------------------------------
// Exit action
	IF (me.StateMachine.intState<>me.StateMachine.intStateNext) THEN
		CIf.Job.intACmd:= cCMD_DONE;
		CIf.Job.intMCmd:= cCMD_DONE;
	END_IF
END_METHOD

{attribute 'object_name' := 'StateMachine'}
METHOD PROTECTED StateMachine : BOOL
SUPER^.StateMachine();

// main statemachine of base controller
CASE me.StateMachine.intState OF
    cBCC_STA_READBusy: 
        THIS^.sta_READBusy();
    cBCC_STA_READ: 
        THIS^.sta_READ();	
END_CASE;
END_METHOD

END_FUNCTION_BLOCK

// POUs/Controller/Lvl0/CYL (Cylinder)/FB_CYL
FUNCTION_BLOCK FB_CYL EXTENDS FB_CtrlBase

VAR_INPUT
	In_bolRetracted: BOOL;
	In_bolExtended: BOOL;
END_VAR
VAR_OUTPUT
	Out_bolRetract: BOOL;
	Out_bolExtend: BOOL;
END_VAR

VAR
	/// Specific interface struct for public access
	SIf: T_Ctrl_SIf_CYL;
END_VAR

(*__________________________________________________________________________________________________
¦	
¦	Vistaprint Schweiz GmbH
¦	CH - 8401 Winterthur
¦
¦	www.vistaprint.ch - info@vistaprint.ch
¦___________________________________________________________________________________________________

Function desription:
Cylinder implementation. 


History:
Version		Date			Author		Comment
---------------------------------------------------------------------------------------------------
0.00.1		25.04.2013		AVME/KVO	Start history
0.00.2		03.07.2013		AVME/KVO	Always call Super.always, no change to off when switch to automatic
										alarm evt EOFF, OFF or cmd off detection in Always
0.00.3		05.11.2013		AVME/KVO	integrate in BaseElements library, 
										FB alarm pointer used, alarm definition over ENUM
0.00.4		17.02.2014		AVME/KVO	Bug fix transission	PON to OFFBusy added	
___________________________________________________________________________________________________*)


SUPER^();

(*
IF (me.bolActivate) THEN // cyclic call enabled
	IF (CIf.Info.bolInitDone=FALSE) THEN // first cycle -> init
		CtrlInit();
		CIf.Info.bolInitDone := TRUE;
	ELSE
		CycleStartDuty();
	
		Always();
		
		StateMachine();
		
		CycleEndDuty();
	END_IF
END_IF;
*)

METHOD PROTECTED Always : BOOL
IF (me.bolChangeBackToAUTO=TRUE) THEN // switch mode to automatic switch off controller
	//me.StateMachine.intStateNext := cSTA_OFFBusy;
	me.bolChangeBackToAUTO := FALSE; // for cylinder no change to off when switch to automatic!!
END_IF

SUPER^.Always();

// ----------------------------------------------------------------------------------
// cyclic actions outside of statemachine
IF (me.StateMachine.intState<>cSTA_SINGLE_ANSWER) THEN
	
	; // always error supervision
	// ----------------------------------------------------------------------------------
	// overrule error always from base -> no EOFF State!! in EOFF go to OFF
	IF (me.StateMachine.intStateNext = cSTA_EOFFBusy) THEN
		IF (me.StateMachine.intState=cSTA_OFF) THEN
			me.StateMachine.intStateNext := cSTA_OFF;
		ELSE // stay in OFF
			me.StateMachine.intStateNext := cSTA_OFFBusy;
		END_IF
	END_IF
END_IF
END_METHOD

METHOD FB_init : BOOL
VAR_INPUT
	///if TRUE, the retain variables are initialized (warm start / cold start)
	bInitRetains: BOOL;
	///if TRUE, the instance afterwards gets moved into the copy code (online change)
	bInCopyCode: BOOL;
END_VAR
VAR
	ii: UINT;
END_VAR
//------------------------------------------------------------------------------------------------------------------------
// to manually change in new FUB implementation!!!
// define valid commands for this controller
FOR ii:= 0 TO (SIZEOF(CIf.Job.aCmdList)/SIZEOF(CIf.Job.aCmdList[0])-1) BY 1 DO
	IF (CIf.Job.aCmdList[ii].intCmd=cCMD_INITIALIZED) THEN
		// found first empty array element
		EXIT;
	END_IF
END_FOR

CIf.Job.aCmdList[ii].intCmd := cCMD_STOP;
CIf.Job.aCmdList[ii].strName := 'Stop'; 
CIf.Job.aCmdList[ii].bolAvailable := TRUE;
ii := ii +1;
CIf.Job.aCmdList[ii].intCmd := cCMD_RETRACT;
CIf.Job.aCmdList[ii].strName := 'Retract';
CIf.Job.aCmdList[ii].bolAvailable := TRUE;
ii := ii +1;
CIf.Job.aCmdList[ii].intCmd := cCMD_EXTEND; // for test simulation single answer
CIf.Job.aCmdList[ii].strName := 'Extend';
CIf.Job.aCmdList[ii].bolAvailable := TRUE;

// set name of class/typ
CIf.Info.strType := 'FB_CYL';
CIf.Info.strFullName := 'Cylinder';

// set alarm class
SIf.Alm[E_ALM_CYL.SensorRetractAlwaysOn].eAlmClass := E_AlmClass.TSTOP;
SIf.Alm[E_ALM_CYL.SensorRetractAlwaysOn].strText := 'sensor retract always on'; 
SIf.Alm[E_ALM_CYL.SensorExtendNotReached].eAlmClass := E_AlmClass.TSTOP;
SIf.Alm[E_ALM_CYL.SensorExtendNotReached].strText := 'timeout extend - sensor extend not reached';
SIf.Alm[E_ALM_CYL.SensorExtendAlwaysOn].eAlmClass := E_AlmClass.TSTOP;
SIf.Alm[E_ALM_CYL.SensorExtendAlwaysOn].strText := 'sensor extend always on';
SIf.Alm[E_ALM_CYL.SensorRetractNotReached].eAlmClass := E_AlmClass.TSTOP;
SIf.Alm[E_ALM_CYL.SensorRetractNotReached].strText := 'timeout retract - sensor retract not reached';
SIf.Alm[E_ALM_CYL.InterlockExtend].eAlmClass := E_AlmClass.OFF;
SIf.Alm[E_ALM_CYL.InterlockExtend].strText := 'interlock extend - movement stopped';
SIf.Alm[E_ALM_CYL.InterlockRetract].eAlmClass := E_AlmClass.OFF;
SIf.Alm[E_ALM_CYL.InterlockRetract].strText := 'interlock retract - movement stopped';

//*******************************************************************************
// initial values
//*******************************************************************************

// Configuration defaults of class
CIf.SwCfg.bolExist := TRUE;
CIf.SwCfg.bolEnable := TRUE;
CIf.SwCfg.bolSimulation := FALSE;

// Parameter defaults of class
SIf.Par.udiExtendTime_ms := 10000;
SIf.Par.udiRetractTime_ms := 8000;
SIf.Par.udiSimExtendTime_ms := SIf.Par.udiExtendTime_ms/2;	
SIf.Par.udiSimRetractTime_ms := SIf.Par.udiRetractTime_ms/2;
END_METHOD

METHOD PROTECTED getCmdState : STRING
VAR_INPUT
	intCmdState: INT;
	bolState: BOOL;
END_VAR
getCmdState := SUPER^.getCmdState(intCmdState:=intCmdState,bolState:=bolState); // get global/base defined cmds/states
IF (getCmdState='') THEN // global not defined get local
	// get string cmd/state string information in runtime
	IF (bolState=FALSE) THEN
		// cmd's
		CASE intCmdState OF
			CYL_CmdState.cCMD_RETRACT: 
				getCmdState := 'cCMD_RETRACT';
			CYL_CmdState.cCMD_EXTEND: 
				getCmdState := 'cCMD_EXTEND';
		ELSE
			getCmdState := 'Cmd not defined';
		END_CASE;
	ELSE
	
	// cmd's
		CASE intCmdState OF
			CYL_CmdState.cSTA_RETRACTBusy: 
				getCmdState := 'cSTA_RETRACTBusy';
			CYL_CmdState.cSTA_RETRACT: 
				getCmdState := 'cSTA_RETRACT';
			CYL_CmdState.cSTA_EXTENDBusy: 
				getCmdState := 'cSTA_EXTENDBusy';
			CYL_CmdState.cSTA_EXTEND: 
				getCmdState := 'cSTA_EXTEND';
		ELSE
			getCmdState := 'State not defined';
		END_CASE;
	END_IF
END_IF
END_METHOD

METHOD getCtrlSIf : POINTER TO T_Ctrl_SIf_CYL
getCtrlSIf := ADR(SIf);
END_METHOD

METHOD PROTECTED IoInBridge : BOOL
// digitale and analoge inputs read from hardware or forcing
SIf.In.bolExtended.map := THIS^.In_bolExtended;
SIf.In.bolRetracted.map := THIS^.In_bolRetracted;

IF (CIf.SwCfg.bolSimulation = FALSE) THEN
	getInBol(CIf.Job.bolIoForce,ADR(SIf.In.bolExtended));
	getInBol(CIf.Job.bolIoForce,ADR(SIf.In.bolRetracted));
ELSE
	//simulation of global IO
END_IF
END_METHOD

METHOD PROTECTED IoOutBridge : BOOL
VAR
	bolSwitchValvesOff: BOOL;
END_VAR
// digitale and analoge inputs read from hardware or forcing
IF (CIf.SwCfg.bolSimulation = FALSE) THEN
	setOutBol(CIf.Job.bolIoForce ,ADR(SIf.Out.bolExtend));
	setOutBol(CIf.Job.bolIoForce ,ADR(SIf.Out.bolRetract));
	
	// check interlocks to prevent damages
	IF (CIf.Job.bolIlkOverwrite=FALSE) THEN
		bolSwitchValvesOff := FALSE;
		
		IF (SIf.Ilk.bolExtend=TRUE) THEN
			// switch off?
			IF (SIf.Cfg.eTyp = E_Typ_CYL.Valve1_Sensor0) OR (SIf.Cfg.eTyp = E_Typ_CYL.Valve1_Sensor2) 
				OR (SIf.Cfg.eTyp = E_Typ_CYL.Valve1_SensorExtended) OR (SIf.Cfg.eTyp = E_Typ_CYL.Valve1_SensorRetracted) THEN
				// monostabil valve -> do nothing
			ELSE
				// bistable valve ->  switch both off
				bolSwitchValvesOff := TRUE;
				IF (SIf.Out.bolExtend.map=1) THEN
					pfbAlarmCtrl^.setAlarm(CIf.Info.intCtrlId,E_ALM_CYL.InterlockExtend,0,ADR(SIf.Alm),E_AlmState.RST,CIf.Job.eMe_ActivAlmClass);
				END_IF
			END_IF
		END_IF
		
		IF (SIf.Ilk.bolRetract=TRUE) THEN
			// switch off?
			IF (SIf.Cfg.eTyp = E_Typ_CYL.Valve1_Sensor0) OR (SIf.Cfg.eTyp = E_Typ_CYL.Valve1_Sensor2) 
				OR (SIf.Cfg.eTyp = E_Typ_CYL.Valve1_SensorExtended) OR (SIf.Cfg.eTyp = E_Typ_CYL.Valve1_SensorRetracted) THEN
				// monostabil valve -> do nothing
				;
			ELSE
				// bistable valve -> switch both off
				bolSwitchValvesOff := TRUE;
				IF (SIf.Out.bolRetract.map=1) THEN
					pfbAlarmCtrl^.setAlarm(CIf.Info.intCtrlId,E_ALM_CYL.InterlockRetract,0,ADR(SIf.Alm),E_AlmState.RST,CIf.Job.eMe_ActivAlmClass);
				END_IF;
			END_IF
		END_IF
		
		// bistable valve -> switch both off
		IF (bolSwitchValvesOff) THEN
			SIf.Out.bolExtend.map := FALSE;
			SIf.Out.bolRetract.map := FALSE;
		END_IF
		
	END_IF

	THIS^.Out_bolExtend := SIf.Out.bolExtend.map;
	THIS^.Out_bolRetract := SIf.Out.bolRetract.map;
END_IF
END_METHOD

METHOD PROTECTED sta_ERROR : BOOL
// state implemetation
//--------------------------------------------------------------------------------------
// Entry action
	IF (me.StateMachine.intState<>me.StateMachine.intStateLastCycle) THEN
		me.StateMachine.intStateHistory := me.StateMachine.intStateLastCycle; // -> possibillity to go back to state before error
		me.StateMachine.intStateLastCycle := me.StateMachine.intState;
		
	END_IF


//--------------------------------------------------------------------------------------
// Cyclic action
	IF (me.StateMachine.intState=me.StateMachine.intStateLastCycle) THEN
		
		;
		
		
		// State Change Condition
		IF (CIf.Job.bolAlmReset = TRUE) THEN
			me.StateMachine.intStateNext := cSTA_ERRORQuit;
		END_IF
	END_IF




//--------------------------------------------------------------------------------------
// Exit action
	IF (me.StateMachine.intState<>me.StateMachine.intStateNext) THEN
		;
	END_IF
END_METHOD

METHOD PROTECTED sta_ERRORQuit : BOOL
// state implemetation
//--------------------------------------------------------------------------------------
// Entry action
	IF (me.StateMachine.intState<>me.StateMachine.intStateLastCycle) THEN
		me.StateMachine.intStateLastCycle := me.StateMachine.intState;
		
	END_IF


//--------------------------------------------------------------------------------------
// Cyclic action
	IF (me.StateMachine.intState=me.StateMachine.intStateLastCycle) THEN
		
		;
		// evtl. wait time if reset of device is necessary and then decide to go to states or ERROR state
		IF (CIf.Job.bolAlmReset = TRUE) THEN
			CIf.Job.eMe_ActivAlmClass := E_AlmClass.NONE; // reset feedback channel for parent
			CIf.Job.bolAlmReset := FALSE;
		END_IF
		
		// State Change Condition
		IF (CIf.Job.bolAlmReset = FALSE) THEN
			IF (me.StateMachine.intStateHistory<=cSTA_PON) THEN
				me.StateMachine.intStateNext := cSTA_PONBusy;
			ELSIF(me.intCmd=cCMD_OFF) THEN
				me.StateMachine.intStateNext := cSTA_OFFBusy;
			ELSIF(me.intCmd=cCMD_STOP) THEN
				me.StateMachine.intStateNext := cSTA_STOPBusy;
			ELSIF(me.intCmd=cCMD_RETRACT) THEN
				me.StateMachine.intStateNext := cSTA_RETRACTBusy;
			ELSIF(me.intCmd=cCMD_EXTEND) THEN
				me.StateMachine.intStateNext := cSTA_EXTENDBusy;
			END_IF
		END_IF
	END_IF


//--------------------------------------------------------------------------------------
// Exit action
	IF (me.StateMachine.intState<>me.StateMachine.intStateNext) THEN
		;
	END_IF
END_METHOD

METHOD PROTECTED sta_EXTEND : BOOL
// state implemetation
//--------------------------------------------------------------------------------------
// Entry action
	IF (me.StateMachine.intState<>me.StateMachine.intStateLastCycle) THEN
		me.StateMachine.intStateLastCycle := me.StateMachine.intState;

	END_IF


//--------------------------------------------------------------------------------------
// Cyclic action
	IF (me.StateMachine.intState=me.StateMachine.intStateLastCycle) THEN

		// Simulation
		IF (CIf.SwCfg.bolSimulation) THEN
			;
		END_IF
		
		// State Change Condition
		IF (SIf.In.bolRetracted.intern) THEN
			// sensor retract always on
			pfbAlarmCtrl^.setAlarm(CIf.Info.intCtrlId,E_ALM_CYL.SensorRetractAlwaysOn,0,ADR(SIf.Alm),E_AlmState.RST,CIf.Job.eMe_ActivAlmClass);
			me.StateMachine.intStateNext :=  cSTA_ERROR;
		ELSIF ((SIf.In.bolExtended.intern = FALSE) AND ((SIf.Cfg.eTyp = E_Typ_CYL.Valve1_SensorExtended) OR (SIf.Cfg.eTyp = E_Typ_CYL.Valve2_SensorExtended))) THEN // wait time until error?
			me.StateMachine.intStateNext := CYL_CmdState.cSTA_EXTENDBusy;
		ELSIF(me.intCmd=cCMD_STOP) THEN
			me.StateMachine.intStateNext := cSTA_STOPBusy;
		ELSIF(me.intCmd=CYL_CmdState.cCMD_RETRACT) THEN
			me.StateMachine.intStateNext := CYL_CmdState.cSTA_RETRACTBusy;
		END_IF
	END_IF



//--------------------------------------------------------------------------------------
// Exit action
	IF (me.StateMachine.intState<>me.StateMachine.intStateNext) THEN
		;
	END_IF
END_METHOD

METHOD PROTECTED sta_EXTENDBusy : BOOL
// state implemetation
//--------------------------------------------------------------------------------------
// Entry action
	IF (me.StateMachine.intState<>me.StateMachine.intStateLastCycle) THEN
		me.StateMachine.intStateLastCycle := me.StateMachine.intState;

		fbSimulationTimer.IN := FALSE;
		fbSimulationTimer.PT := UDINT_TO_TIME(SIf.Par.udiSimExtendTime_ms);
		fbSimulationTimer(); // set time/reset timer
		fbSimulationTimer.IN := TRUE; // start timer
	END_IF


//--------------------------------------------------------------------------------------
// Cyclic action
	IF (me.StateMachine.intState=me.StateMachine.intStateLastCycle) THEN

		// Simulation
		IF (CIf.SwCfg.bolSimulation) THEN
			fbSimulationTimer(); // simulation time
			IF (fbSimulationTimer.Q) THEN
				SIf.In.bolExtended.intern := TRUE;
				SIf.In.bolRetracted.intern := FALSE;
			END_IF
		END_IF
		
		//no change action
		SIf.Out.bolExtend.intern := TRUE;
		SIf.Out.bolRetract.intern := FALSE;
		
		
		// State Change Condition
		IF (me.StateMachine.udiTimeInState_ms>SIf.Par.udiExtendTime_ms) THEN
			IF (SIf.In.bolRetracted.intern) THEN
				// sensor retract always on
				pfbAlarmCtrl^.setAlarm(CIf.Info.intCtrlId,E_ALM_CYL.SensorRetractAlwaysOn,0,ADR(SIf.Alm),E_AlmState.RST,CIf.Job.eMe_ActivAlmClass);
			ELSE
				// timeout extend
				pfbAlarmCtrl^.setAlarm(CIf.Info.intCtrlId,E_ALM_CYL.SensorExtendNotReached,0,ADR(SIf.Alm),E_AlmState.RST,CIf.Job.eMe_ActivAlmClass);
			END_IF
			me.StateMachine.intStateNext :=  cSTA_ERROR;
		ELSIF (SIf.In.bolExtended.intern) AND (SIf.In.bolRetracted.intern=FALSE) THEN
			me.StateMachine.intStateNext := CYL_CmdState.cSTA_EXTEND;
		ELSIF ((SIf.Cfg.eTyp = E_Typ_CYL.Valve1_SensorRetracted) OR (SIf.Cfg.eTyp = E_Typ_CYL.Valve2_SensorRetracted))
				 AND (SIf.In.bolRetracted.intern=FALSE) AND (me.StateMachine.udiTimeInState_ms>SIf.Par.udiSimExtendTime_ms) THEN
			me.StateMachine.intStateNext := CYL_CmdState.cSTA_EXTEND;
		ELSIF ((SIf.Cfg.eTyp = E_Typ_CYL.Valve1_Sensor0) OR (SIf.Cfg.eTyp = E_Typ_CYL.Valve2_Sensor0))
				AND (me.StateMachine.udiTimeInState_ms>SIf.Par.udiSimExtendTime_ms) THEN
			me.StateMachine.intStateNext := CYL_CmdState.cSTA_EXTEND;		
		ELSIF(me.intCmd=cCMD_STOP) THEN
			me.StateMachine.intStateNext := cSTA_STOPBusy;
		ELSIF(me.intCmd=cCMD_RETRACT) THEN
			me.StateMachine.intStateNext := CYL_CmdState.cSTA_RETRACTBusy;
		END_IF
	END_IF




//--------------------------------------------------------------------------------------
// Exit action
	IF (me.StateMachine.intState<>me.StateMachine.intStateNext) THEN
		SIf.Cur.udiMoveTimeExtend := me.StateMachine.udiTimeInState_ms;
	END_IF
END_METHOD

METHOD PROTECTED sta_OFF : BOOL
// state implemetation
//--------------------------------------------------------------------------------------
// Entry action
	IF (me.StateMachine.intState<>me.StateMachine.intStateLastCycle) THEN
		me.StateMachine.intStateLastCycle := me.StateMachine.intState;
		
	END_IF


//--------------------------------------------------------------------------------------
// Cyclic action
	IF (me.StateMachine.intState=me.StateMachine.intStateLastCycle) THEN
		
		;
		
		// State Change Condition
		IF (me.Alarm.eActivAlmClass<>E_AlmClass.EOFF) AND (me.Alarm.eActivAlmClass<>E_AlmClass.OFF) THEN
			IF (me.intCmd=cCMD_STOP) THEN
				// sensor retract always on cylinder
				me.StateMachine.intStateNext :=  cSTA_STOPBusy;
			ELSIF (me.intCmd=CYL_CmdState.cCMD_EXTEND) THEN 
				me.StateMachine.intStateNext := cSTA_EXTENDBusy;
			ELSIF(me.intCmd=CYL_CmdState.cCMD_RETRACT) THEN
				me.StateMachine.intStateNext := cSTA_RETRACTBusy;
			END_IF
		END_IF
	END_IF




//--------------------------------------------------------------------------------------
// Exit action
	IF (me.StateMachine.intState<>me.StateMachine.intStateNext) THEN
		;
	END_IF
END_METHOD

METHOD PROTECTED sta_OFFBusy : BOOL
// state implemetation
//--------------------------------------------------------------------------------------
// Entry action
	IF (me.StateMachine.intState<>me.StateMachine.intStateLastCycle) THEN
		me.StateMachine.intStateLastCycle := me.StateMachine.intState;
		
	END_IF


//--------------------------------------------------------------------------------------
// Cyclic action
	IF (me.StateMachine.intState=me.StateMachine.intStateLastCycle) THEN
		
		// switch off?
		IF (SIf.Cfg.eTyp = E_Typ_CYL.Valve1_Sensor0) OR (SIf.Cfg.eTyp = E_Typ_CYL.Valve1_Sensor2) 
			OR (SIf.Cfg.eTyp = E_Typ_CYL.Valve1_SensorExtended) OR (SIf.Cfg.eTyp = E_Typ_CYL.Valve1_SensorRetracted) THEN
			// monostabil valve -> do nothing
			;
		ELSE
			// bistable valve -> switch both off
			SIf.Out.bolExtend.intern := FALSE;
			SIf.Out.bolRetract.intern := FALSE;
		END_IF
		
		
		
		// State Change Condition
		IF (TRUE) THEN
			me.StateMachine.intStateNext := cSTA_OFF;
		END_IF
	END_IF




//--------------------------------------------------------------------------------------
// Exit action
	IF (me.StateMachine.intState<>me.StateMachine.intStateNext) THEN
		;
	END_IF
END_METHOD

METHOD PROTECTED sta_RETRACT : BOOL
// state implemetation
//--------------------------------------------------------------------------------------
// Entry action
	IF (me.StateMachine.intState<>me.StateMachine.intStateLastCycle) THEN
		me.StateMachine.intStateLastCycle := me.StateMachine.intState;

	END_IF


//--------------------------------------------------------------------------------------
// Cyclic action
	IF (me.StateMachine.intState=me.StateMachine.intStateLastCycle) THEN

		// Simulation
		IF (CIf.SwCfg.bolSimulation) THEN
			;
		END_IF
		
		// State Change Condition
		IF (SIf.In.bolExtended.intern) THEN
			// sensor retract always on
			pfbAlarmCtrl^.setAlarm(CIf.Info.intCtrlId,E_ALM_CYL.SensorExtendAlwaysOn,0,ADR(SIf.Alm),E_AlmState.RST,CIf.Job.eMe_ActivAlmClass);
			me.StateMachine.intStateNext :=  cSTA_ERROR;
		ELSIF ((SIf.In.bolRetracted.intern = FALSE) AND ((SIf.Cfg.eTyp = E_Typ_CYL.Valve1_SensorRetracted) OR (SIf.Cfg.eTyp = E_Typ_CYL.Valve2_SensorRetracted))) THEN // wait time until error?
			me.StateMachine.intStateNext := CYL_CmdState.cSTA_RETRACTBusy;
		ELSIF(me.intCmd=cCMD_STOP) THEN
			me.StateMachine.intStateNext := cSTA_STOPBusy;
		ELSIF(me.intCmd=CYL_CmdState.cCMD_EXTEND) THEN
			me.StateMachine.intStateNext := CYL_CmdState.cSTA_EXTENDBusy;
		END_IF
	END_IF




//--------------------------------------------------------------------------------------
// Exit action
	IF (me.StateMachine.intState<>me.StateMachine.intStateNext) THEN
		;
	END_IF
END_METHOD

METHOD PROTECTED sta_RETRACTBusy : BOOL
// state implemetation
//--------------------------------------------------------------------------------------
// Entry action
	IF (me.StateMachine.intState<>me.StateMachine.intStateLastCycle) THEN
		me.StateMachine.intStateLastCycle := me.StateMachine.intState;
		
		SIf.Out.bolExtend.intern := FALSE;
		SIf.Out.bolRetract.intern := TRUE;
		
		fbSimulationTimer.IN := FALSE;
		fbSimulationTimer.PT := UDINT_TO_TIME(SIf.Par.udiSimRetractTime_ms);
		fbSimulationTimer(); // set time/reset timer
		fbSimulationTimer.IN := TRUE; // start timer
	END_IF


//--------------------------------------------------------------------------------------
// Cyclic action
	IF (me.StateMachine.intState=me.StateMachine.intStateLastCycle) THEN

		// Simulation
		IF (CIf.SwCfg.bolSimulation) THEN
			fbSimulationTimer(); // simulation time
			IF (fbSimulationTimer.Q) THEN
				SIf.In.bolRetracted.intern := TRUE;
				SIf.In.bolExtended.intern := FALSE;
			END_IF
		END_IF
		
		// State Change Condition
		IF (me.StateMachine.udiTimeInState_ms>SIf.Par.udiRetractTime_ms) THEN
			IF (SIf.In.bolExtended.intern) THEN
				// sensor extend always on 
				pfbAlarmCtrl^.setAlarm(CIf.Info.intCtrlId,E_ALM_CYL.SensorExtendAlwaysOn,0,ADR(SIf.Alm),E_AlmState.RST,CIf.Job.eMe_ActivAlmClass);
			ELSE
				// timeout retract cylinder
				pfbAlarmCtrl^.setAlarm(CIf.Info.intCtrlId,E_ALM_CYL.SensorRetractNotReached,0,ADR(SIf.Alm),E_AlmState.RST,CIf.Job.eMe_ActivAlmClass);
			END_IF
			me.StateMachine.intStateNext :=  cSTA_ERROR;
		ELSIF (SIf.In.bolRetracted.intern) AND(SIf.In.bolExtended.intern=FALSE) THEN
			me.StateMachine.intStateNext := CYL_CmdState.cSTA_RETRACT;
		ELSIF ((SIf.Cfg.eTyp = E_Typ_CYL.Valve1_SensorExtended) OR (SIf.Cfg.eTyp = E_Typ_CYL.Valve2_SensorExtended))
				 AND (SIf.In.bolExtended.intern=FALSE) AND (me.StateMachine.udiTimeInState_ms>SIf.Par.udiSimRetractTime_ms) THEN
			me.StateMachine.intStateNext := CYL_CmdState.cSTA_RETRACT;
		ELSIF ((SIf.Cfg.eTyp = E_Typ_CYL.Valve1_Sensor0) OR (SIf.Cfg.eTyp = E_Typ_CYL.Valve2_Sensor0))
				AND (me.StateMachine.udiTimeInState_ms>SIf.Par.udiSimRetractTime_ms) THEN
			me.StateMachine.intStateNext := CYL_CmdState.cSTA_RETRACT;		
		ELSIF(me.intCmd=cCMD_STOP) THEN
			me.StateMachine.intStateNext := cSTA_STOPBusy;
		ELSIF(me.intCmd=CYL_CmdState.cCMD_EXTEND) THEN
			me.StateMachine.intStateNext := CYL_CmdState.cSTA_EXTENDBusy;
		END_IF
	END_IF




//--------------------------------------------------------------------------------------
// Exit action
	IF (me.StateMachine.intState<>me.StateMachine.intStateNext) THEN
		SIf.Cur.udiMoveTimeRetract := me.StateMachine.udiTimeInState_ms;
	END_IF
END_METHOD

METHOD PROTECTED sta_STOP : BOOL
// state implemetation
//--------------------------------------------------------------------------------------
// Entry action
	IF (me.StateMachine.intState<>me.StateMachine.intStateLastCycle) THEN
		me.StateMachine.intStateLastCycle := me.StateMachine.intState;
		
	END_IF


//--------------------------------------------------------------------------------------
// Cyclic action
	IF (me.StateMachine.intState=me.StateMachine.intStateLastCycle) THEN
		
		;
		
		
		// State Change Condition
		IF (me.intCmd=CYL_CmdState.cCMD_EXTEND) THEN 
			me.StateMachine.intStateNext := CYL_CmdState.cSTA_EXTENDBusy;
		ELSIF(me.intCmd=CYL_CmdState.cCMD_RETRACT) THEN
			me.StateMachine.intStateNext := CYL_CmdState.cSTA_RETRACTBusy;
		END_IF
	END_IF




//--------------------------------------------------------------------------------------
// Exit action
	IF (me.StateMachine.intState<>me.StateMachine.intStateNext) THEN
		;
	END_IF
END_METHOD

METHOD PROTECTED sta_STOPBusy : BOOL
// state implemetation
//--------------------------------------------------------------------------------------
// Entry action
	IF (me.StateMachine.intState<>me.StateMachine.intStateLastCycle) THEN
		me.StateMachine.intStateLastCycle := me.StateMachine.intState;
		
	END_IF


//--------------------------------------------------------------------------------------
// Cyclic action
	IF (me.StateMachine.intState=me.StateMachine.intStateLastCycle) THEN
		
		// switch off?
		IF (SIf.Cfg.eTyp = E_Typ_CYL.Valve1_Sensor0) OR (SIf.Cfg.eTyp = E_Typ_CYL.Valve1_Sensor2) 
			OR (SIf.Cfg.eTyp = E_Typ_CYL.Valve1_SensorExtended) OR (SIf.Cfg.eTyp = E_Typ_CYL.Valve1_SensorRetracted) THEN
			// monostabil valve -> do nothing
			;
		ELSE
			// bistable valve -> switch both on -> block at position
			SIf.Out.bolExtend.intern := TRUE;
			SIf.Out.bolRetract.intern := TRUE;
		END_IF
		
		
		
		// State Change Condition
		IF (TRUE) THEN
			me.StateMachine.intStateNext := cSTA_STOP;
		END_IF
	END_IF




//--------------------------------------------------------------------------------------
// Exit action
	IF (me.StateMachine.intState<>me.StateMachine.intStateNext) THEN
		;
	END_IF
END_METHOD

METHOD PROTECTED StateMachine : BOOL
SUPER^.StateMachine();

// main statemachine of base controller
CASE me.StateMachine.intState OF
    CYL_CmdState.cSTA_RETRACTBusy: 
        THIS^.sta_RETRACTBusy();
    CYL_CmdState.cSTA_RETRACT: 
        THIS^.sta_RETRACT();
    CYL_CmdState.cSTA_EXTENDBusy: 
        THIS^.sta_EXTENDBusy();
    CYL_CmdState.cSTA_EXTEND: 
        THIS^.sta_EXTEND();
	cSTA_STOPBusy: 
        THIS^.sta_STOPBusy();
    cSTA_STOP: 
        THIS^.sta_STOP();
END_CASE;
END_METHOD

END_FUNCTION_BLOCK

// POUs/Controller/Lvl0/DRV (Drive)/FB_DRV
FUNCTION_BLOCK FB_DRV EXTENDS FB_CtrlBase
VAR_INPUT
	In_bolOverload: BOOL;
	In_bolPulse: BOOL;
	In_a_bolBlockedSupvervis: ARRAY[1..cMAX_BLOCKED_SUP] OF BOOL;
	In_bolMaintenanceSwitch: BOOL;
END_VAR
VAR_OUTPUT
	Out_bolSpeed_1: BOOL;
	Out_bolSpeed_2: BOOL;
END_VAR
VAR
	/// Specific interface struct for public access
	SIf: T_Ctrl_SIf_DRV;
	bolPulseFlag: BOOL;
	udiPulseTimeoutTimer: UDINT;
	/// Timer for speed average calculation
	udiTimerSpeedCalc: UDINT;
	/// Shift register for average calculation of the speed
	aSpeedShift: ARRAY[0..4] OF DINT;
	/// Size of Speed Shift array for average calculation
	intSpeedShiftSize: INT;
	/// Varible for Speedcalculation
	dinSpeedCalc_um_s: DINT;
	/// Varible for Speedcalculation
	dinSpeedNew_um_s: DINT;
	/// Old Position for Speed calculation
	dinPosOld_um: DINT;
	/// Loop variable
	intI: INT;
	/// Blocked supervision
	/// Array with supervision distances
	a_dintPinDistance: ARRAY[1..cMAX_BLOCKED_SUP] OF DINT;
	a_bolREBlockedSupvervis: ARRAY[1..cMAX_BLOCKED_SUP] OF BOOL;
	/// Old Position for from last cycle
	dinPosOldCycle_um: DINT;
END_VAR
VAR CONSTANT
	/// Check speed every 250ms
	cSpeedCalcTime_ms: UDINT := 250;
END_VAR

(*__________________________________________________________________________________________________
¦	
¦	Vistaprint Schweiz GmbH
¦	CH - 8401 Winterthur
¦
¦	www.vistaprint.ch - info@vistaprint.ch
¦___________________________________________________________________________________________________

Function desription:
Drive element for all different Drive types, 
Configuration of the type and Speed Calculation


History:
Version		Date			Author		Comment
---------------------------------------------------------------------------------------------------
0.00.1		27.06.2013		VP/RE		Start history
0.00.2		28.08.2013		AVME/PRE	Implement speed calculation
0.00.3		19.09.2013		AVME/PRE	Implement new Base Concept
0.00.4		02.10.2013		VP/RE		Added pulse counter. Changed pulse distance to 28.4 mm as a default value. Changed driving distance to 305 mm.
0.00.5      10.10.2013		AVME/DSC    In_bolBufferFull deleted. Not needed in DRV controller. Handled by parent controller if necessary.
0.00.6      18.10.2013		AVME/DSC    SIf.Alm[4].strText deleted in FB_init. Not used anymore.
0.00.7		22.10.2013		AVME/MRU	DRV without pulse sensor simulated pulse imroved
0.00.8      23.10.2013		AVME/DSC    Speed calculation from always to state RUN. cSpeedCalcTime_ms -> 250ms. Shift register array 0..4. Clear buffer in state RUN entry action.
										Changes for better position interpolation in controllers like MER, DPJ, DHC and JUN.
0.00.9		09.07.2014		AVME/MRU	Add Maintenance Switch to Drive (Used in Windsor)
										
___________________________________________________________________________________________________*)


SUPER^();

(*
IF (me.bolActivate) THEN // cyclic call enabled
	IF (CIf.Info.bolInitDone=FALSE) THEN // first cycle -> init
		CtrlInit();
		CIf.Info.bolInitDone := TRUE;
	ELSE
		CycleStartDuty();
	
		Always();
		
		StateMachine();
		
		CycleEndDuty();
	END_IF
END_IF;
*)

METHOD PROTECTED Always : BOOL
SUPER^.Always();

IF (me.StateMachine.intState<>cSTA_SINGLE_ANSWER) THEN
	
	// Error checks not in OFF and Error States
	IF (me.StateMachine.intState<>cSTA_OFF) AND (me.StateMachine.intState<>cSTA_ERROR) AND (me.StateMachine.intState<>cSTA_ERRORQuit) THEN

		IF (SIf.Cfg.bolEnableMaintenaceSwitch AND SIf.In.bolMaintenanceSwitch.intern) THEN
			// SIf.Alm[4].strText := 'Maintenance Switch is OFF'; 
			pfbAlarmCtrl^.setAlarm(CIf.Info.intCtrlId,4,0,ADR(SIf.Alm),E_AlmState.RST,CIf.Job.eMe_ActivAlmClass);		
			me.StateMachine.intStateNext := cSTA_ERROR;		
		END_IF

		IF SIf.In.bolOverload.intern THEN
			// SIf.Alm[1].strText := 'Drive overload'; 
			pfbAlarmCtrl^.setAlarm(CIf.Info.intCtrlId,1,0,ADR(SIf.Alm),E_AlmState.RST,CIf.Job.eMe_ActivAlmClass);		
			me.StateMachine.intStateNext := cSTA_ERROR;		
		END_IF
		
		// Blocked Supervision control
		// Sensor detect Pins, if a defined count of pins are brocken, the machine stops
		FOR intI := 1 TO SIf.Cfg.usiCountBlockedSupervis DO
			
			// Simulation
			// Simulate the Pins in the drive
			IF (CIf.SwCfg.bolSimulation) THEN
				IF (a_dintPinDistance[intI] >  SIf.Cfg.dinPinDistance_um) THEN
					SIf.In.a_bolBlockedSupvervis[intI].intern := TRUE;
				ELSE
					SIf.In.a_bolBlockedSupvervis[intI].intern := FALSE;
				END_IF
			END_IF
		
			// Check if a new pin is arrive, set distance to last pin to '0'
			IF ((SIf.In.a_bolBlockedSupvervis[intI].intern = TRUE) AND (a_bolREBlockedSupvervis[intI] = FALSE)) THEN
				a_bolREBlockedSupvervis[intI] := TRUE;
				a_dintPinDistance[intI] := 0;
			ELSIF ((SIf.In.a_bolBlockedSupvervis[intI].intern = FALSE) AND (a_bolREBlockedSupvervis[intI] = TRUE)) THEN
				a_bolREBlockedSupvervis[intI] := FALSE;
			END_IF
			// Check distance to last Pin, if to far away, set error
			IF (a_dintPinDistance[intI] > ((SIf.Par.int_MaxBrokenPins+1) * SIf.Cfg.dinPinDistance_um)) THEN
				// SIf.Alm[3].strText := 'Drive blocked, Pins are broken'; 
				pfbAlarmCtrl^.setAlarm(CIf.Info.intCtrlId,3,0,ADR(SIf.Alm),E_AlmState.RST,CIf.Job.eMe_ActivAlmClass);
				a_dintPinDistance[intI] := 0;		
				me.StateMachine.intStateNext := cSTA_ERROR;		
			ELSE
				a_dintPinDistance[intI] := a_dintPinDistance[intI] + SIf.Cur.dinPos_um - dinPosOldCycle_um;					
			END_IF		
		END_FOR
		dinPosOldCycle_um := SIf.Cur.dinPos_um;
	END_IF
END_IF

// Speed calculation in always function to get correct position everytime, not only in run
// observe no pulse detected failure case 
IF (SIf.In.bolPulse.intern AND NOT(bolPulseFlag)) THEN				
	// calculate CUR
	SIf.Cur.dinPos_um := SIf.Cur.dinPos_um + SIf.Cfg.dinDistPerPulse_um;
	SIf.Cur.dinPulseCounter := SIf.Cur.dinPulseCounter + 1;
		
	udiPulseTimeoutTimer := 0;
	bolPulseFlag := TRUE;
ELSIF (NOT(SIf.In.bolPulse.intern) AND bolPulseFlag) THEN
	bolPulseFlag := FALSE;
END_IF

// Always change actions in Base Library
// ----------------------------------------------------------------------------------
// overrule error always from base -> no EOFF State!! in EOFF go to OFF
IF (me.StateMachine.intStateNext = cSTA_EOFFBusy) THEN
	IF (me.StateMachine.intState=cSTA_OFF) THEN
		me.StateMachine.intStateNext := cSTA_OFF;
	ELSE // stay in OFF
		me.StateMachine.intStateNext := cSTA_OFFBusy;
	END_IF
END_IF
END_METHOD

METHOD FB_init : BOOL
VAR_INPUT
	///if TRUE, the retain variables are initialized (warm start / cold start)
	bInitRetains: BOOL;
	///if TRUE, the instance afterwards gets moved into the copy code (online change)
	bInCopyCode: BOOL;
END_VAR
VAR
	ii: UINT;
END_VAR
//------------------------------------------------------------------------------------------------------------------------
// to manually change in new FUB implementation!!!
// define valid commands for this controller
FOR ii:= 0 TO (SIZEOF(CIf.Job.aCmdList)/SIZEOF(CIf.Job.aCmdList[0])-1) BY 1 DO
	IF (CIf.Job.aCmdList[ii].intCmd=cCMD_INITIALIZED) THEN
		// found first empty array element
		EXIT;
	END_IF
END_FOR
CIf.Job.aCmdList[ii].intCmd := cCMD_RUN;
CIf.Job.aCmdList[ii].strName := 'Run'; 
CIf.Job.aCmdList[ii].bolAvailable := TRUE;
ii := ii +1;

// set name of class/typ
CIf.Info.strType := 'FB_DRV';
CIf.Info.strFullName := 'Drive';

// set alarm class
SIf.Alm[1].eAlmClass := E_AlmClass.OFF;
SIf.Alm[1].strText := 'Drive overload'; 
SIf.Alm[2].eAlmClass := E_AlmClass.OFF;
SIf.Alm[2].strText := 'Timeout no pulse detected';
SIf.Alm[3].eAlmClass := E_AlmClass.OFF;
SIf.Alm[3].strText := 'Drive blocked, Pins are broken';
SIf.Alm[4].eAlmClass := E_AlmClass.OFF;
SIf.Alm[4].strText := 'Maintenance Switch is OFF'; 

//*******************************************************************************
// initial values
//*******************************************************************************

// software configuration
CIf.SwCfg.bolExist := TRUE;
CIf.SwCfg.bolSimulation := FALSE;

// parmeter
SIf.Par.udi_pulseTimeout_ms := 2000;
SIf.Par.udi_pulseSim_ms := 56;
SIf.Par.usi_speedLevel := 0;
SIf.Par.int_MaxBrokenPins := 5;

SIf.Cfg.dinDistPerPulse_um := 28400; // 28,4[mm/puls]
SIf.Cfg.usiCountBlockedSupervis := 0;
SIf.Cfg.dinPinDistance_um := 305000;
SIf.Cfg.bolEnableMaintenaceSwitch := FALSE; // Normaly no Maintenance Switch exist
END_METHOD

METHOD getCtrlSIf : POINTER TO T_Ctrl_SIf_DRV
getCtrlSIf := ADR(SIf);
END_METHOD

METHOD PROTECTED IoInBridge : BOOL
// digitale and analoge inputs read from hardware or forcing
SIf.In.bolOverload.map := THIS^.In_bolOverload;
SIf.In.bolPulse.map := THIS^.In_bolPulse;
SIf.In.bolMaintenanceSwitch.map := THIS^.In_bolMaintenanceSwitch;

FOR intI := 1 TO SIf.Cfg.usiCountBlockedSupervis DO
	SIf.In.a_bolBlockedSupvervis[intI].map := THIS^.In_a_bolBlockedSupvervis[intI];
	IF (CIf.SwCfg.bolSimulation = FALSE) THEN
		getInBol(CIf.Job.bolIoForce,ADR(SIf.In.a_bolBlockedSupvervis[intI]));
	END_IF
END_FOR

IF (CIf.SwCfg.bolSimulation = FALSE) THEN
	getInBol(CIf.Job.bolIoForce,ADR(SIf.In.bolOverload));
	getInBol(CIf.Job.bolIoForce,ADR(SIf.In.bolPulse));
	//ctrl.In.bol_PosSwitchBasicDefTyp.intern := getInBol(ctrl.ifc.Job.bol_Force ,ADR(ctrl.In.bol_PosSwitchBasicDefTyp);
	getInBol(CIf.Job.bolIoForce,ADR(SIf.In.bolMaintenanceSwitch));
ELSE
	//simulation of global IO
	SIf.In.bolOverload.intern := FALSE;
	SIf.In.bolMaintenanceSwitch.intern := FALSE;
END_IF
END_METHOD

METHOD PROTECTED IoOutBridge : BOOL
VAR
	bolSwitchValvesOff: BOOL;
END_VAR
// digitale and analoge inputs read from hardware or forcing
IF (CIf.SwCfg.bolSimulation = FALSE) THEN
	setOutBol(CIf.Job.bolIoForce ,ADR(SIf.Out.bolSpeed_1));
	setOutBol(CIf.Job.bolIoForce ,ADR(SIf.Out.bolSpeed_2));

	THIS^.Out_bolSpeed_1 := SIf.Out.bolSpeed_1.map;
	THIS^.Out_bolSpeed_2 := SIf.Out.bolSpeed_2.map;
END_IF
END_METHOD

METHOD PRIVATE SetSpeed
// 0=slow, 1=middle, 2=fast
CASE SIf.Par.usi_speedLevel OF
	0:
		SIf.Out.bolSpeed_1.intern := TRUE;
		SIf.Out.bolSpeed_2.intern := FALSE;
	1:
		SIf.Out.bolSpeed_1.intern := TRUE;
		SIf.Out.bolSpeed_2.intern := TRUE;
	2:
		SIf.Out.bolSpeed_1.intern := FALSE;
		SIf.Out.bolSpeed_2.intern := TRUE;
	ELSE
		SIf.Out.bolSpeed_1.intern := TRUE;
		SIf.Out.bolSpeed_2.intern := FALSE;
END_CASE
END_METHOD

METHOD PROTECTED sta_ERROR : BOOL
// state implemetation
//--------------------------------------------------------------------------------------
// Entry action
IF (me.StateMachine.intState<>me.StateMachine.intStateLastCycle) THEN
	me.StateMachine.intStateHistory := me.StateMachine.intStateLastCycle; // -> possibillity to go back to state before error
	me.StateMachine.intStateLastCycle := me.StateMachine.intState;
	
	SIf.Out.bolSpeed_1.intern := FALSE;
	SIf.Out.bolSpeed_2.intern := FALSE;
	
END_IF


//--------------------------------------------------------------------------------------
// Cyclic action
	IF (me.StateMachine.intState=me.StateMachine.intStateLastCycle) THEN
		
		;
		
		
		// State Change Condition
		IF (CIf.Job.bolAlmReset = TRUE) THEN
			me.StateMachine.intStateNext := cSTA_ERRORQuit;
		END_IF
	END_IF




//--------------------------------------------------------------------------------------
// Exit action
	IF (me.StateMachine.intState<>me.StateMachine.intStateNext) THEN
		;
	END_IF
END_METHOD

METHOD PROTECTED sta_OFF : BOOL
// state implemetation
//--------------------------------------------------------------------------------------
// Entry action
	IF (me.StateMachine.intState<>me.StateMachine.intStateLastCycle) THEN
		me.StateMachine.intStateLastCycle := me.StateMachine.intState;
		
	END_IF


//--------------------------------------------------------------------------------------
// Cyclic action
	IF (me.StateMachine.intState=me.StateMachine.intStateLastCycle) THEN
		
		;
		
		
		// State Change Condition
		IF (me.Alarm.eActivAlmClass<>E_AlmClass.EOFF) AND (me.Alarm.eActivAlmClass<>E_AlmClass.OFF) THEN
			IF (me.intCmd=cCMD_RUN) THEN 
				me.StateMachine.intStateNext := cSTA_RUNBusy;
			END_IF
		END_IF
	END_IF




//--------------------------------------------------------------------------------------
// Exit action
	IF (me.StateMachine.intState<>me.StateMachine.intStateNext) THEN
		;
	END_IF
END_METHOD

METHOD PROTECTED sta_OFFBusy : BOOL
// state implemetation
//--------------------------------------------------------------------------------------
// Entry action
	IF (me.StateMachine.intState<>me.StateMachine.intStateLastCycle) THEN
		me.StateMachine.intStateLastCycle := me.StateMachine.intState;
		
	END_IF


//--------------------------------------------------------------------------------------
// Cyclic action
	IF (me.StateMachine.intState=me.StateMachine.intStateLastCycle) THEN
		
		SIf.Out.bolSpeed_1.intern := FALSE;
		SIf.Out.bolSpeed_2.intern := FALSE;
		
		// State Change Condition
		IF (TRUE) THEN
			me.StateMachine.intStateNext := cSTA_OFF;
		END_IF
	END_IF




//--------------------------------------------------------------------------------------
// Exit action
	IF (me.StateMachine.intState<>me.StateMachine.intStateNext) THEN
		;
	END_IF
END_METHOD

METHOD PROTECTED sta_PON : BOOL
// state implemetation
//--------------------------------------------------------------------------------------
// Entry action
	IF (me.StateMachine.intState<>me.StateMachine.intStateLastCycle) THEN
		me.StateMachine.intStateLastCycle := me.StateMachine.intState;
		
	END_IF


//--------------------------------------------------------------------------------------
// Cyclic action
	IF (me.StateMachine.intState=me.StateMachine.intStateLastCycle) THEN
		
		;
		
		
		// State Change Condition
		IF ((me.intCmd=cCMD_OFF) OR (me.intCmd=cCMD_RUN)) THEN
			me.StateMachine.intStateNext := cSTA_OFFBusy;
		END_IF
	END_IF




//--------------------------------------------------------------------------------------
// Exit action
	IF (me.StateMachine.intState<>me.StateMachine.intStateNext) THEN
		;
	END_IF
END_METHOD

METHOD PROTECTED sta_RUN : BOOL
VAR
	ii: INT;
END_VAR
// state implemetation
//--------------------------------------------------------------------------------------
// Entry action
	IF (me.StateMachine.intState<>me.StateMachine.intStateLastCycle) THEN
		me.StateMachine.intStateLastCycle := me.StateMachine.intState;
		
		udiPulseTimeoutTimer := 0;
		bolPulseFlag := FALSE;
		
		fbSimulationTimer.IN := FALSE;
		fbSimulationTimer.PT := UDINT_TO_TIME(SIf.Par.udi_pulseSim_ms);  
		fbSimulationTimer(); // set time/reset timer
		fbSimulationTimer.IN := TRUE; // start timer
			
		// Get Size of array
		intSpeedShiftSize := SIZEOF(aSpeedShift)/(SIZEOF(aSpeedShift[0]));
		// Clear speed buffer
		FOR ii:=0 TO intSpeedShiftSize-1 BY 1 DO
			aSpeedShift[ii]:=0;
		END_FOR
		
	END_IF


//--------------------------------------------------------------------------------------
// Cyclic action
	IF (me.StateMachine.intState=me.StateMachine.intStateLastCycle) THEN
		
		// Simulation
		// AND speed simulation if no distance sensor is existing !!!
		IF ((CIf.SwCfg.bolSimulation) OR (SIf.Cfg.bolPulseExist = FALSE)) THEN
			fbSimulationTimer(); // simulation time
			IF (fbSimulationTimer.Q) THEN
				SIf.In.bolPulse.intern := TRUE; 
				In_bolPulse := TRUE; // MRU 22.10.2013 added for drive without pulse sensor
				fbSimulationTimer.IN := FALSE;
			ELSE
				SIf.In.bolPulse.intern := FALSE;
				In_bolPulse := FALSE; // MRU 22.10.2013 added for drive without pulse sensor
				fbSimulationTimer.IN := TRUE;
			END_IF
		END_IF
	
		IF SIf.Cfg.bolSpeedVariable = TRUE THEN
			SetSpeed();
		END_IF;
		
		udiPulseTimeoutTimer := udiPulseTimeoutTimer + me.FUBInfo.udiSample_ms;
		
		
		// Speed calculation
		IF udiTimerSpeedCalc >= cSpeedCalcTime_ms THEN
			dinSpeedNew_um_s := (SIf.Cur.dinPos_um - dinPosOld_um)*1000 / UDINT_TO_DINT(udiTimerSpeedCalc);
			dinSpeedCalc_um_s := dinSpeedNew_um_s;
			// Get Size of array
			intSpeedShiftSize := SIZEOF(aSpeedShift)/(SIZEOF(aSpeedShift[0]));
			intI := intSpeedShiftSize-1;
			WHILE intI > 0 DO		
				// Shift all speeds one field
				aSpeedShift[intI] := aSpeedShift[intI-1];
				dinSpeedCalc_um_s := dinSpeedCalc_um_s + aSpeedShift[intI];
				intI := intI - 1;
			END_WHILE
			aSpeedShift[0] := dinSpeedNew_um_s;
			SIf.Cur.dinSpeed_um_s := dinSpeedCalc_um_s / intSpeedShiftSize;
			dinPosOld_um := SIf.Cur.dinPos_um;
			udiTimerSpeedCalc := 0;
				
		ELSE
			udiTimerSpeedCalc := udiTimerSpeedCalc + me.FUBInfo.udiSample_ms;
		END_IF
		
		
		// State Change Condition
		IF ((udiPulseTimeoutTimer >= Sif.Par.udi_pulseTimeout_ms) AND (SIf.Cfg.bolPulseExist = TRUE)) THEN
			// SIf.Alm[2].strText := 'Timeout no pulse detected';
			pfbAlarmCtrl^.setAlarm(CIf.Info.intCtrlId,2,0,ADR(SIf.Alm),E_AlmState.RST,CIf.Job.eMe_ActivAlmClass);

			me.StateMachine.intStateNext :=  cSTA_ERROR;		
		ELSIF (me.intCmd=cCMD_OFF) THEN
			me.StateMachine.intStateNext :=  cSTA_OFFBusy;
		END_IF
		
	END_IF



//--------------------------------------------------------------------------------------
// Exit action
	IF (me.StateMachine.intState<>me.StateMachine.intStateNext) THEN
		// Set speed zero
		SIf.Cur.dinSpeed_um_s := 0;
	END_IF
END_METHOD

METHOD PROTECTED sta_RUNBusy : BOOL
// state implemetation
//--------------------------------------------------------------------------------------
// Entry action
	IF (me.StateMachine.intState<>me.StateMachine.intStateLastCycle) THEN
		me.StateMachine.intStateLastCycle := me.StateMachine.intState;
		
	END_IF


//--------------------------------------------------------------------------------------
// Cyclic action
	IF (me.StateMachine.intState=me.StateMachine.intStateLastCycle) THEN

		IF SIf.Cfg.bolSpeedVariable = TRUE THEN
			SetSpeed();
		ELSE
			SIf.Out.bolSpeed_1.intern := TRUE;
		END_IF;		
		
		// State Change Condition
		IF (TRUE) THEN
			me.StateMachine.intStateNext := cSTA_RUN;
		END_IF
	END_IF




//--------------------------------------------------------------------------------------
// Exit action
	IF (me.StateMachine.intState<>me.StateMachine.intStateNext) THEN
		;
	END_IF
END_METHOD

METHOD PROTECTED StateMachine : BOOL
SUPER^.StateMachine();

// main statemachine of base controller
CASE me.StateMachine.intState OF
    cSTA_RUNBusy: 
        THIS^.sta_RUNBusy();
    cSTA_RUN: 
        THIS^.sta_RUN();
END_CASE;
END_METHOD

END_FUNCTION_BLOCK

// POUs/Controller/Lvl0/ECD (EtherCAT Diagnostic)/FB_ECD
FUNCTION_BLOCK FB_ECD EXTENDS FB_CtrlBase
VAR
	/// Specific interface struct for public access
	SIf: T_Ctrl_SIf_ECD;
	/// Number State Errors in this cycle
	udiNumOfStateErrors: UDINT;
	/// Number CRC Errors in this cycle
	udiNumOfCRCErrors: UDINT;
	/// Loop variable for request
	uinLoop: UINT;
	/// Loop variable for Slaves
	uinLoopSlave: UINT;
	/// Number of Slaves for internal use
	uinSlaveNbr: UINT;
	/// Variable to calculat the error information
	dinAlarmInfo: DINT;
	/// Feedback from functions
	bolFBbusy: BOOL;
	/// Save The Reset of CRC Errors
	bolResetCRCError: BOOL;
	/// Feedback from functions
	bolFBerror: BOOL;
	udiFBerror: UDINT;
	/// Array of all Adresses
	arrSlaveAdress: ARRAY[0..ECD_Const.cuinMaxSlaves] OF UINT;
	/// Array of all Slave Data
	arrSlaveConf: ARRAY[0..ECD_Const.cuinMaxSlaves] OF Tc2_EtherCAT.ST_EcSlaveConfigData;
	/// Array of Abnormal State Changes
	arrSlaveAbnormalStates: ARRAY[0..ECD_Const.cuinMaxSlaves] OF UDINT;
	/// Number of configurated Slaves
	uinConfigSlaveNbr: UINT;
	/// Slavenumber internal
	uinErrorSlaveAdr: UINT;
	/// Numbers of Slave Errors
	uinErrorSlaveNbr: UINT;
	/// Information of Error
	uinErrorSlaveInfo: UINT;
	/// Adress of Link Error
	uinErrorSlaveLink: UINT;
	/// Numbers of Link Error
	uinErrorSlaveLinkNbr: UINT;
	/// Information of Link Error
	uinErrorSlaveLinkInfo: UINT;
	/// Slavenumber internal
	uinErrorSlaveAdrCRC: UINT;
	/// Numbers of Slave Errors
	uinErrorSlaveNbrCRC: UINT;
	/// Information of Error
	uinErrorSlaveInfoCRC: UINT;
	/// Internal Alarmtextes to insert additional informations
	arrAlmtexts: ARRAY[1..(E_ALM_ECD.MAX_E_ALM - 1)] OF STRING;
	strAlarminfo: STRING;
	/// Functional Blocks
	fbEcGetAllSlaveAddr: Tc2_EtherCAT.FB_EcGetAllSlaveAddr;
	fbEcGetConfSlaves: Tc2_EtherCAT.FB_EcGetConfSlaves;
	fbEcGetMasterState: Tc2_EtherCAT.FB_EcGetMasterState;
	fbEcGetSlaveState: Tc2_EtherCAT.FB_EcGetSlaveState;
	fbEcGetSlaveCrcError: Tc2_EtherCAT.FB_EcGetSlaveCrcErrorEx;
	fbEcGetAllSlaveAbnormalStateChanges: Tc2_EtherCAT.FB_EcGetAllSlaveAbnormalStateChanges;
	fbEcMasterFrameStatisticClearCRC: Tc2_EtherCAT.FB_EcMasterFrameStatisticClearCRC;
END_VAR
VAR CONSTANT
	/// Sub states
	cSTA_SUB_INITIALIZE: INT := 500;
	cSTA_SUB_GetAllSlaveAdress: INT := 501;
	cSTA_SUB_GetAllSlaveAdressDone: INT := 502;
	cSTA_SUB_GetConfSlaves: INT := 503;
	cSTA_SUB_GetConfSlavesDone: INT := 504;
	cSTA_SUB_CheckMaster: INT := 505;
	cSTA_SUB_CheckMasterDone: INT := 506;
	cSTA_SUB_CheckSlaveChanges: INT := 507;
	cSTA_SUB_CheckSlaveChangesDone: INT := 508;
	cSTA_SUB_SLAVE_START: INT := 509;
	cSTA_SUB_CheckSlaveState: INT := 510;
	cSTA_SUB_CheckSlaveStateDone: INT := 511;
	cSTA_SUB_CheckCRC: INT := 512;
	cSTA_SUB_CheckCRCDone: INT := 513;
	cSTA_SUB_CheckCRCReset: INT := 514;
	cSTA_SUB_CheckCRCResetDone: INT := 515;
	cSTA_SUB_Inc: INT := 516;
	cSTA_SUB_WAIT_NEXT_POLL: INT := 517;
	cSTA_SUB_ERROR: INT := 560;
	cSTA_SUB_DONE: INT := 520;
END_VAR

(*__________________________________________________________________________________________________
¦	
¦	Vistaprint Schweiz GmbH
¦	CH - 8401 Winterthur
¦
¦	www.vistaprint.ch - info@vistaprint.ch
¦___________________________________________________________________________________________________

Function desription:
EtherCAT Diagnostics for Hardware and communication errors
Diagnosis of the EtherCAT with Beckhoff FUB's to check if there are some errors in the network 

History:
Version		Date			Author		Comment
---------------------------------------------------------------------------------------------------
0.00.1		25.04.2014		AVME/PRE	Start history

___________________________________________________________________________________________________*)

SUPER^();

(*
IF (me.bolActivate) THEN // cyclic call enabled
	IF (CIf.Info.bolInitDone=FALSE) THEN // first cycle -> init
		CtrlInit();
		CIf.Info.bolInitDone := TRUE;
	ELSE
		CycleStartDuty();
	
		Always();
		
		StateMachine();
		
		CycleEndDuty();
	END_IF
END_IF;
*)

METHOD PROTECTED Always : BOOL
SUPER^.Always();

// ----------------------------------------------------------------------------------
// cyclic actions outside of statemachine
IF (me.StateMachine.intState<>cSTA_SINGLE_ANSWER) THEN
	;	
END_IF


// ----------------------------------------------------------------------------------
// Always change actions in Base Library
// ----------------------------------------------------------------------------------
// overrule error always from base -> no EOFF State!! in EOFF go to OFF
IF (me.StateMachine.intStateNext = cSTA_EOFFBusy) THEN
	IF (me.StateMachine.intState=cSTA_OFF) THEN
		me.StateMachine.intStateNext := cSTA_OFF;
	ELSE // stay in OFF
		me.StateMachine.intStateNext := cSTA_OFFBusy;
	END_IF
END_IF
END_METHOD

METHOD FB_init : BOOL
VAR_INPUT
	///if TRUE, the retain variables are initialized (warm start / cold start)
	bInitRetains: BOOL;
	///if TRUE, the instance afterwards gets moved into the copy code (online change)
	bInCopyCode: BOOL;
END_VAR
VAR
	udiTaskCnt: UDINT;
	ii: UINT;
END_VAR
//------------------------------------------------------------------------------------------------------------------------
// to manually change in new FUB implementation!!!
// define valid commands for this controller
FOR ii:= 0 TO (SIZEOF(CIf.Job.aCmdList)/SIZEOF(CIf.Job.aCmdList[0])-1) BY 1 DO
	IF (CIf.Job.aCmdList[ii].intCmd=cCMD_INITIALIZED) THEN
		// found first empty array element
		EXIT;
	END_IF
END_FOR
CIf.Job.aCmdList[ii].intCmd := cCMD_RUN;
CIf.Job.aCmdList[ii].strName := 'Run'; 
CIf.Job.aCmdList[ii].bolAvailable := TRUE;
ii := ii +1;

// set name of class/typ
CIf.Info.strType := 'FB_ECD';
CIf.Info.strFullName := 'EtherCAT Diagnostic';

// set alarm class
SIf.Alm[E_ALM_ECD.ADS_ComError].eAlmClass := E_AlmClass.INFO;
SIf.Alm[E_ALM_ECD.ADS_ComError].strText := 'ADS Communication Error to EtherCAT Master'; // ADS Communication Error to EtherCAT Master => Info = ADS_Errorcode
SIf.Alm[E_ALM_ECD.TimeOutFunction].eAlmClass := E_AlmClass.INFO;
SIf.Alm[E_ALM_ECD.TimeOutFunction].strText := 'Timeout EtherCAT function'; // A Function is not finished after the defined Timeout
SIf.Alm[E_ALM_ECD.NotAllSlaveConnected].eAlmClass := E_AlmClass.OFF;
SIf.Alm[E_ALM_ECD.NotAllSlaveConnected].strText := 'Not all configurated Slaves Found ';// Configured and reached Slaves are not the same => Info Byte 0+1 = Slave Addres from last error Info Byte 2+3 = Numbers of error Slaves
SIf.Alm[E_ALM_ECD.ToManySlaves].eAlmClass := E_AlmClass.INFO;
SIf.Alm[E_ALM_ECD.ToManySlaves].strText := 'To many slaves';// More slaves at the master as the structure could handle => Info Byte 0+1 = Slave Addres from last error Info Byte 2+3 = Numbers of error Slaves
SIf.Alm[E_ALM_ECD.MasterStateError].eAlmClass := E_AlmClass.OFF;
SIf.Alm[E_ALM_ECD.MasterStateError].strText := 'Master State Error'; // Master not in the correct state => Info = Masterstate
SIf.Alm[E_ALM_ECD.SlaveStateError].eAlmClass := E_AlmClass.INFO;
SIf.Alm[E_ALM_ECD.SlaveStateError].strText := 'Slave State Error'; // Minimum one Slave not in the correct state => Byte 0+1 = Slave Addres from first error, Info Byte 2 + 3 = State of first error Slave
SIf.Alm[E_ALM_ECD.SlaveCRCError].eAlmClass := E_AlmClass.INFO;
SIf.Alm[E_ALM_ECD.SlaveCRCError].strText :=  'Slave CRC Error';	// Minimum one Slave has to many CRC Erros => Byte 0+1 = Slave Addres from first error or the one with the most CRC errors, Info Byte 2 + 3 = Number of CRC Errors from first Slave with error
SIf.Alm[E_ALM_ECD.SlaveLinkError].eAlmClass := E_AlmClass.INFO;
SIf.Alm[E_ALM_ECD.SlaveLinkError].strText :=  'Slave Link State Error'; // Minimum one Slave has a LinkState Erros => Byte 0+1 = Slave Addres from first error Info Byte 2 + 3 = Link State of first error Slave
SIf.Alm[E_ALM_ECD.NoSlaveFound].eAlmClass := E_AlmClass.INFO;
SIf.Alm[E_ALM_ECD.NoSlaveFound].strText :=  'No Slave in Network'; 		// No EtherCAT Slave found in the network
SIf.Alm[E_ALM_ECD.StateChanges].eAlmClass := E_AlmClass.INFO;
SIf.Alm[E_ALM_ECD.StateChanges].strText :=  'To many Abnormal State Changes'; 		// No EtherCAT Slave found in the network

//*******************************************************************************
// initial values
//*******************************************************************************

// software configuration
CIf.SwCfg.bolExist := TRUE;
CIf.SwCfg.bolSimulation := FALSE;

// parameter
SIf.Par.udiTOCheckOne_ms:= 1500;
SIf.Par.udiTOCheckAll_ms:= 5000;
SIf.Par.udiTOPowerOn_ms:= 10000;
SIf.Par.udiPollingInterval_ms:= 10000;
SIf.Par.udiMaxCRC:= 50;
END_METHOD

METHOD PROTECTED getCmdState : STRING
VAR_INPUT
	intCmdState: INT;
	bolState: BOOL;
END_VAR
getCmdState := SUPER^.getCmdState(intCmdState:=intCmdState,bolState:=bolState); // get global/base defined cmds/states
IF (getCmdState='') THEN // global not defined get local
	// get string cmd/state string information in runtime
	IF (bolState=FALSE) THEN
		(*
		// cmd's
		CASE intCmdState OF
			;
		END_CASE
		*)
	ELSE
		// states
		CASE intCmdState OF
			// SUB States
			cSTA_SUB_INITIALIZE:
				getCmdState := 'cSTA_SUB_INITIALIZE';
			cSTA_SUB_GetAllSlaveAdress:
				getCmdState := 'cSTA_SUB_GetAllSlaveAdress';
			cSTA_SUB_GetAllSlaveAdressDone:
				getCmdState := 'cSTA_SUB_GetAllSlaveAdressDone';
			cSTA_SUB_GetConfSlaves:
				getCmdState := 'cSTA_SUB_GetConfSlaves';
			cSTA_SUB_GetConfSlavesDone:
				getCmdState := 'cSTA_SUB_GetConfSlavesDone';			
			cSTA_SUB_CheckMaster:
				getCmdState := 'cSTA_SUB_CheckMaster';	
			cSTA_SUB_CheckMasterDone:
				getCmdState := 'cSTA_SUB_CheckMasterDone';	
			cSTA_SUB_CheckSlaveChanges:
				getCmdState := 'cSTA_SUB_CheckSlaveChanges';	
			cSTA_SUB_CheckSlaveChangesDone:
				getCmdState := 'cSTA_SUB_CheckSlaveChangesDone';				
			cSTA_SUB_SLAVE_START:
				getCmdState := 'cSTA_SUB_SLAVE_START';				
			cSTA_SUB_CheckSlaveState:
				getCmdState := 'cSTA_SUB_CheckSlaveState';	
			cSTA_SUB_CheckSlaveStateDone:
				getCmdState := 'cSTA_SUB_CheckSlaveStateDone';	
			cSTA_SUB_CheckCRC:
				getCmdState := 'cSTA_SUB_CheckCRC';	
			cSTA_SUB_CheckCRCDone:
				getCmdState := 'cSTA_SUB_CheckCRCDone';	
			cSTA_SUB_CheckCRCReset:
				getCmdState := 'cSTA_SUB_CheckCRCReset';	
			cSTA_SUB_CheckCRCResetDone:
				getCmdState := 'cSTA_SUB_CheckCRCResetDone';	
			cSTA_SUB_Inc:
				getCmdState := 'cSTA_SUB_Inc';	
		
			cSTA_SUB_ERROR:
				getCmdState := 'cSTA_SUB_ERROR';
			cSTA_SUB_DONE:
				getCmdState := 'cSTA_SUB_DONE';
			cSTA_SUB_WAIT_NEXT_POLL:
				getCmdState := 'cSTA_SUB_WAIT_NEXT_POLL';
				

		END_CASE
	END_IF
END_IF
END_METHOD

METHOD getCtrlSIf : POINTER TO T_Ctrl_SIf_ECD
getCtrlSIf := ADR(SIf);
END_METHOD

METHOD PROTECTED sta_ERROR : BOOL
// state implemetation
//--------------------------------------------------------------------------------------
// Entry action
	IF (me.StateMachine.intState<>me.StateMachine.intStateLastCycle) THEN
		me.StateMachine.intStateHistory := me.StateMachine.intStateLastCycle; // -> possibillity to go back to state before error
		me.StateMachine.intStateLastCycle := me.StateMachine.intState;
		
		// Initialize sub state machine
		me.SubStateMachine.intState:= cSTA_SUB_INITIALIZE; 
		me.SubStateMachine.intStateNext := cSTA_SUB_INITIALIZE;
	END_IF

//--------------------------------------------------------------------------------------
// Cyclic action
	IF (me.StateMachine.intState=me.StateMachine.intStateLastCycle) THEN
		// State Change Condition
		IF (CIf.Job.bolAlmReset = TRUE) THEN
			me.StateMachine.intStateNext := cSTA_ERRORQuit;
		END_IF
	END_IF

//--------------------------------------------------------------------------------------
// Exit action
	IF (me.StateMachine.intState<>me.StateMachine.intStateNext) THEN
		;
	END_IF
END_METHOD

METHOD PROTECTED sta_ERRORQuit : BOOL
// state implemetation
//--------------------------------------------------------------------------------------
// Entry action
	IF (me.StateMachine.intState<>me.StateMachine.intStateLastCycle) THEN
		me.StateMachine.intStateLastCycle := me.StateMachine.intState;
		// Prepare Function Block
		bolResetCRCError := TRUE;
		fbEcMasterFrameStatisticClearCRC(sNetId:= SIf.Cfg.strNetID, 
										bExecute:= FALSE, 
										tTimeout:= UDINT_TO_TIME(SIf.Par.udiTOCheckAll_ms));
				
		// Start Function
		fbEcMasterFrameStatisticClearCRC(bExecute:= TRUE, 
										tTimeout:= UDINT_TO_TIME(SIf.Par.udiTOCheckAll_ms));
		
	END_IF


//--------------------------------------------------------------------------------------
// Cyclic action
	IF (me.StateMachine.intState=me.StateMachine.intStateLastCycle) THEN
		
		;
		// evtl. wait time if reset of device is necessary and then decide to go to states or ERROR state
		IF (CIf.Job.bolAlmReset = TRUE) THEN
			CIf.Job.eMe_ActivAlmClass := E_AlmClass.NONE; // reset feedback channel for parent
			CIf.Job.bolAlmReset := FALSE;
		END_IF
		// **************************************************************************
		// Wait until Reset all CRC Error is Done
		// **************************************************************************
			fbEcMasterFrameStatisticClearCRC(bExecute:= FALSE);
			// Wait until done
			IF NOT (fbEcMasterFrameStatisticClearCRC.bBusy) THEN
				IF NOT (fbEcMasterFrameStatisticClearCRC.bError) THEN
					bolResetCRCError := FALSE;
				// Error
				ELSE
					// SIf.Alm[E_ALM_ECD.ADS_ComError].strText := 'ADS Communication Error to EtherCAT Master'; // ADS Communication Error to EtherCAT Master => Info = ADS_Errorcode
					pfbAlarmCtrl^.setAlarm(CIf.Info.intCtrlId,E_ALM_ECD.ADS_ComError,UDINT_TO_DINT(fbEcGetSlaveCrcError.nErrId),ADR(SIf.Alm),E_AlmState.RST,CIf.Job.eMe_ActivAlmClass);
					me.StateMachine.intStateNext := cSTA_SUB_ERROR;		
				END_IF
			END_IF
		
